	(* Falls nur Zentrierung aktiviert ist, dann zuerst den Schnellhub stoppen *)
	50:	IF NOT(xStFct_InitStep) THEN
			xStFct_InitStep:=TRUE;
			IF gxOnlyCentringActive OR (wStFct_Status = 99) OR (wStFct_Status = 1) OR (wStFct_Status = 98) THEN
				IF (T_Station_Parameter.T_StProcess.rCentringSpeedOAxis > 0.0) THEN
					QxFastStrokeOn_St1:=FALSE;
					QiAFastStroke:=0;
					TONWaitStopOAxis(IN:=FALSE,PT:=T#0.5s);
				ELSE
					TONWaitStopOAxis(IN:=FALSE,PT:=T#0.01s);
				END_IF;
			ELSE
				TONWaitStopOAxis(IN:=FALSE,PT:=T#0.01s);
			END_IF;
		END_IF;
		TONWaitStopOAxis(IN:=TRUE);
		IF TONWaitStopOAxis.Q THEN
			TONWaitStopOAxis(IN:=FALSE);
			xStFct_StartMainPrc:=FALSE;
			xStFct_InitStep:=FALSE;
			iStFct_StepPrc:=iStFct_StepPrc + 1;
		END_IF;
	(* Z1 Achse auf LadePosition zurückfahren ODER einen Offset zurückfahren *)
	51:	IF NOT(xStFct_InitStep) THEN
			xStFct_InitStep:=TRUE;
			IF gxOnlyCentringActive OR (wStFct_Status = 99) OR (wStFct_Status = 1) OR (wStFct_Status = 98) THEN
				ptrTAxisZ^.T_CtrleSingle.iFunction:=7;
				ptrTAxisZ^.T_CtrleSingle.lrPosition:=grZ_LoadPos;
				ptrTAxisZ^.T_CtrleSingle.lrVelocity:=T_Station_Parameter.T_StProcess.rOutfeedStrokeAxisSpeed;
				ptrTAxisZ^.T_CtrleSingle.xExecute:=TRUE;
				IF NOT(ptrTAxisBubbler^.T_CtrleDCAxis.xNotMoving) THEN
					(* Abstreifer ZU *)
					QxCylStripperClose_St1:=TRUE;
					QxCylStripperOpen_St1:=FALSE;
				END_IF
				IF (T_Station_Parameter.T_StProcess.rCentringSpeedOAxis > 0.0) THEN
					QxFastStrokeOn_St1:=FALSE;
					QiAFastStroke:=0;
				END_IF;
			ELSE
				lrZCheckPosition:=ptrTAxisZ^.T_LiveValue.lrActualPosition + T_Station_Parameter.T_StProcess.rCentringOffsetBackward;
				IF (lrZCheckPosition <= grZ_WorkStartPos) THEN
					ptrTAxisZ^.T_CtrleSingle.iFunction:=7;	(* Absolute Bewegung *)
					ptrTAxisZ^.T_CtrleSingle.lrPosition:=grZ_WorkStartPos;
				ELSE
					ptrTAxisZ^.T_CtrleSingle.iFunction:=8;	(* Relative Bewegung *)
					ptrTAxisZ^.T_CtrleSingle.lrDistance:=T_Station_Parameter.T_StProcess.rCentringOffsetBackward;
				END_IF;
				ptrTAxisZ^.T_CtrleSingle.lrVelocity:=T_Station_Parameter.T_StProcess.rCentringBackStrokeSpeed;
				ptrTAxisZ^.T_CtrleSingle.xExecute:=TRUE;
			END_IF;
		END_IF;
		IF (gxOnlyCentringActive OR (wStFct_Status = 99) OR (wStFct_Status = 1) OR (wStFct_Status = 98)) AND (ptrTAxisZ^.T_LiveValue.lrActualPosition <= (garCentringEndProcCalc[1] + T_Station_Parameter.T_StProcess.rCentringOffsetBackward)) THEN
			QxCylWPUnfix_St1:=FALSE;
		END_IF
		IF NOT(ptrTAxisZ^.T_CtrleSingle.xExecute) AND ptrTAxisZ^.T_CtrleSingle.xDone THEN
			xStFct_StartMainPrc:=FALSE;
			xStFct_InitStep:=FALSE;
			iStFct_StepPrc:=iStFct_StepPrc + 1;
			QxCylWPUnfix_St1:=FALSE;
		END_IF;
	(* S Achse stoppen *)
	(* O Achse stoppen *)
	(* ZylWPUnfix zurücksetzen *)
	52:	IF NOT(xStFct_InitStep) THEN
			xStFct_InitStep:=TRUE;
			IF gxOnlyCentringActive OR (wStFct_Status = 99) OR (wStFct_Status = 1) OR (wStFct_Status = 98) THEN
				IF (NOT(ptrTAxisS^.T_CtrleSingle.xNotMoving) OR NOT(ptrTAxisS^.T_CtrleSingle.xDone))
				AND NOT((ptrTAxisS^.T_CtrleSingle.iFunction = 5) AND NOT(ptrTAxisS^.T_CtrleSingle.xDone)) AND NOT(ptrTAxisS^.T_CtrleSingle.xErr) THEN
					ptrTAxisS^.T_CtrleSingle.iFunction:=5;
					ptrTAxisS^.T_CtrleSingle.xExecute:=TRUE;
				END_IF;
				IF (T_Station_Parameter.T_StProcess.rCentringSpeedOAxis > 0.0) THEN
					QxFastStrokeOn_St1:=FALSE;
					QiAFastStroke:=0;
				END_IF;
				QxCylWPUnfix_St1:=FALSE;
			END_IF
			IF xProcessDone THEN
				IF (NOT(ptrTAxisS^.T_CtrleSingle.xNotMoving) OR NOT(ptrTAxisS^.T_CtrleSingle.xDone))
				AND NOT((ptrTAxisS^.T_CtrleSingle.iFunction = 5) AND NOT(ptrTAxisS^.T_CtrleSingle.xDone)) AND NOT(ptrTAxisS^.T_CtrleSingle.xErr) THEN
					ptrTAxisS^.T_CtrleSingle.iFunction:=5;
					ptrTAxisS^.T_CtrleSingle.xExecute:=TRUE;
				END_IF;
				QxFastStrokeOn_St1:=FALSE;
				QiAFastStroke:=0;
			END_IF
			(* Abstreifer AUF *)
			QxCylStripperClose_St1:=FALSE;
			QxCylStripperOpen_St1:=TRUE;
		END_IF;
		IF NOT(ptrTAxisS^.T_CtrleSingle.xExecute) AND ptrTAxisS^.T_CtrleSingle.xDone THEN
			xStFct_StartMainPrc:=FALSE;
			xStFct_InitStep:=FALSE;
			IF (wStFct_Status <> 1) THEN
				iStFct_StepPrc:=90;
			ELSIF (wStFct_Status = 1) THEN
				xStFct_HardwareError:=TRUE;
				diStFct_TmpErrorNr:=41;		(* Zentrierproz. HC1 eingetroffen *)
				RETURN;
			ELSE
				xStFct_HardwareError:=TRUE;
				diStFct_TmpErrorNr:=42;		(* Zentrierproz. StartPos erreicht und HC2 immer noch ON *)
			END_IF;
		END_IF;

	90:	IF gxHardwareOFF OR gxAxisOFF THEN
		(* Gilt nur falls HW ausgeschaltet ist *)
			IF NOT(xStFct_InitStep) THEN
				xStFct_InitStep:=TRUE;
				TONWorkTime(IN:=FALSE);
			END_IF;
			TONWorkTime(IN:=TRUE,PT:=T#5s);
			T_Station_Work.THWWorkStation.TCtrlWork.iOverLimitCounterCentering:=5;
			IF TONWorkTime.Q THEN
				TONWorkTime(IN:=FALSE);
				xStFct_StartMainPrc:=FALSE;
				xStFct_InitStep:=FALSE;
				iStFct_StepPrc:=0;
				xStFct_SetEnd:=TRUE;
				wStFct_Status:=0;
				IF T_Station_Parameter.T_StProcess.xCentringEndProcIncOnOff THEN
					garCentringEndProcCalc[1]:=garCentringEndProcCalc[1] + T_Station_Parameter.T_StProcess.rCentringEndProInc;	(* Zentrier EndPos Inkrementieren *)
				END_IF;
			END_IF;
		ELSE
			xStFct_StartMainPrc:=FALSE;
			xStFct_InitStep:=FALSE;
			iStFct_StepPrc:=0;
			xStFct_SetEnd:=TRUE;
		END_IF;
	END_CASE;
END_IF;
(******************************************************************************************************************************************)
(****************************			             Stationsfunktion Parallelablauf                                       *****************************)
(******************************************************************************************************************************************)
IF xStFct_StartPrc_Parallel AND NOT(xStFct_SetEnd) AND NOT(xStFct_HardwareError) THEN
	CASE iStFct_StepPrc_Parallel OF
	1:	iStFct_StepPrc_Parallel:=1;
		xStFct_InitStep_Parallel:=FALSE;
		xStFct_StartPrc_Parallel:=FALSE;
	END_CASE;
END_IF;
(******************************************************************************************************************************************)
(****************************				     Stationsfunktion Endprozedur                                    *****************************)
(******************************************************************************************************************************************)
StationFunction_Ctrl_End;
END_ACTION

(* POU GENERAL/FB_CalcCuttingSpeed, ST *)
FUNCTION_BLOCK FB_CalcCuttingSpeed
VAR_INPUT
	rActualPosition : REAL;
	iCountStep : INT;	(* Durchschnitt von diesem Counter wird berechnet *)
END_VAR
VAR_IN_OUT
	xCapturePosition : BOOL;
	xReset : BOOL;
END_VAR
VAR_OUTPUT
	rCuttingSpeed : REAL;
END_VAR
VAR
	arCuttingSpeed: ARRAY [1..2,1..200] OF REAL;
	arDeleteData: ARRAY [1..2,1..200] OF REAL;
	iStepCounter: INT;
	rSumDeltaPos : REAL;
	rSumDeltaTime : REAL;
	ii: INT;
	iStepPos: INT;
	xFirstCycle: BOOL;
	rTmpSavePosition: REAL;
	TONCycleTime: TON;
	xStartTimer: BOOL;
	rTmpSaveTime: REAL;
	iTmpStepCount: INT;
END_VAR
(* Berechnung der Schnittgeschwindigkeit *)
IF xReset THEN
	xReset:=FALSE;
	xFirstCycle:=TRUE;
	xStartTimer:=FALSE;
	rCuttingSpeed:=0.0;
	arCuttingSpeed:=arDeleteData;
END_IF;
TONCycleTime(IN:=xStartTimer,PT:=T#999999s);
IF xCapturePosition THEN
	xCapturePosition:=xStartTimer:=FALSE;
	IF xFirstCycle THEN
		iTmpStepCount:=iCountStep;
		IF (iTmpStepCount <= 0) THEN
			iTmpStepCount:=1;
		ELSIF (iTmpStepCount > 200) THEN
			iTmpStepCount:=200;
		END_IF;
		xFirstCycle:=FALSE;
		iStepCounter:=iStepPos:=1;
		rCuttingSpeed:=0.0;
		rTmpSavePosition:=rActualPosition;
		xStartTimer:=TRUE;
		RETURN;
	END_IF;
	rTmpSavePosition:=rActualPosition - rTmpSavePosition;			(* Delta Position *)
	rTmpSaveTime:=TIME_TO_REAL(TONCycleTime.ET)/1000.0;		(* Delta Time *)
	arCuttingSpeed[1,iStepCounter]:=rTmpSavePosition;
	arCuttingSpeed[2,iStepCounter]:=rTmpSaveTime;
	rTmpSavePosition:=rActualPosition;
	rSumDeltaPos:=rSumDeltaTime:=0.0;
	FOR ii:=1 TO iStepPos DO
		rSumDeltaPos:=rSumDeltaPos + arCuttingSpeed[1,ii];
		rSumDeltaTime:=rSumDeltaTime + arCuttingSpeed[2,ii];
	END_FOR;
	rCuttingSpeed:=(rSumDeltaPos/INT_TO_REAL(iStepPos))/(rSumDeltaTime/INT_TO_REAL(iStepPos));
	iStepCounter:=iStepCounter + 1;
	IF (iStepCounter > iTmpStepCount) THEN
		iStepCounter:=1;
	END_IF;
	IF (iStepPos < iTmpStepCount) THEN
		iStepPos:=iStepPos + 1;
	END_IF;
ELSE
	IF NOT(xFirstCycle) THEN
		xStartTimer:=TRUE;
	END_IF;
END_IF;
END_FUNCTION_BLOCK

(* POU GENERAL/FB_SparkOutProcess, ST *)
FUNCTION_BLOCK FB_SparkOutProcess
VAR_INPUT
	lrHubLength: LREAL;
	iCountHub: INT;
	T_Station_Parameter: ST_RETAIN_DATA_STATIONWORK;
	xToolDeflection : BOOL;
	xToolTorqueHC : BOOL;
	xToolTorqueSparkOut : BOOL;
END_VAR
VAR_IN_OUT
	xStart: BOOL;
	xReset: BOOL;
	TCylToolDeflection : ST_CYLINDER;
	TAxisZ : ST_AXIS;
END_VAR
VAR_OUTPUT
	xEnd: BOOL;
	xBlockProcess: BOOL;
	xRepeatProcess: BOOL;
	wStatus: WORD;
	rLastOverLimitPosition: REAL;
	xBlockOutput:BOOL;
	xBlockDeflectionOutput:BOOL;
END_VAR
VAR
	xTmpStart: BOOL;
	xInit: BOOL;
	iStepCounter: INT;
	xInitStep: BOOL;
	lrSaveSlidePosition: LREAL;
	iTmpCountHub: INT;
	xSetForceDeflection: BOOL;
	xInitSetForceDeflection: BOOL;
	xActiveChgForceDeflection: BOOL;
	xBlockCounter: BOOL;
END_VAR
IF xReset THEN
	xReset:=FALSE;
	xEnd:=TRUE;
	xStart:=FALSE;
	xTmpStart:=FALSE;
	xInit:=FALSE;
	xBlockProcess:=FALSE;
	xRepeatProcess:=FALSE;
	xInitStep:=FALSE;
	iTmpCountHub:=0;
	xBlockOutput:=FALSE;
	RETURN;
END_IF;
IF xStart OR xTmpStart THEN
	IF NOT(xInit) THEN
		iStepCounter:=1;
		iTmpCountHub:=0;
		xInit:=TRUE;
		xStart:=FALSE;
		xTmpStart:=TRUE;
		lrSaveSlidePosition:=TAxisZ.T_LiveValue.lrActualPosition;
		xBlockProcess:=xRepeatProcess:=FALSE;
	END_IF;
	CASE iStepCounter OF
		1:	IF NOT(xInitStep) THEN
				xInitStep:=TRUE;
				xBlockProcess:=TRUE;
				xBlockCounter:=FALSE;
				IF (iCountHub > 0) AND (lrHubLength <> 0) THEN
					IF (T_Station_Parameter.T_StProcess.rSparkOutForceDeflection <> 0.0) THEN xActiveChgForceDeflection:=TRUE; ELSE xActiveChgForceDeflection:=FALSE; END_IF;
					IF NOT(xActiveChgForceDeflection) THEN
						xInitStep:=FALSE;
						iStepCounter:=iStepCounter + 1;
						RETURN;
					END_IF;
					IF xActiveChgForceDeflection THEN
						xBlockDeflectionOutput:=TRUE;
						xSetForceDeflection:=TRUE;
						TCylToolDeflection.T_CtrleCyl.T_Analog.rForceIn:=(T_Station_Parameter.T_OnlineChange.rForceDeflection/100.0) * T_Station_Parameter.T_StProcess.rSparkOutForceDeflection;
					ELSE
						xSetForceDeflection:=FALSE;
					END_IF;
				ELSE
					xEnd:=TRUE;
					xInit:=FALSE;
					xInitStep:=FALSE;
					xTmpStart:=FALSE;
					xBlockProcess:=xRepeatProcess:=xBlockOutput:=xBlockDeflectionOutput:=FALSE;
					RETURN;
				END_IF;
			END_IF;
			IF NOT(xSetForceDeflection) THEN
				xInitStep:=FALSE;
				iStepCounter:=iStepCounter + 1;
			END_IF;
		2:	IF NOT(xInitStep) THEN
				xInitStep:=TRUE;
				(* Move Absolut backward or forward *)
				TAxisZ.T_CtrleSingle.iFunction:=7;
				TAxisZ.T_CtrleSingle.lrPosition:=TAxisZ.T_LiveValue.lrActualPosition + lrHubLength;
				TAxisZ.T_CtrleSingle.lrAcceleration:=TAxisZ.T_Config_ObjFileValue.lrAcceleration;
				TAxisZ.T_CtrleSingle.lrDecceleration:=TAxisZ.T_Config_ObjFileValue.lrDecceleration;
				TAxisZ.T_CtrleSingle.lrJerk:=TAxisZ.T_Config_ObjFileValue.lrJerk;
				TAxisZ.T_CtrleSingle.lrVelocity:=T_Station_Parameter.T_StProcess.rSparkOutStrokeSpeed;
				TAxisZ.T_CtrleSingle.xExecute:=TRUE;
			END_IF;
			IF TAxisZ.T_CtrleSingle.xMovingForward THEN
				IF xToolDeflection THEN
					wStatus:=1;	(* 1 = < Wz Auslenk. Sensor > *)
					xInitStep:=FALSE;
					iStepCounter:=iStepCounter + 2;
					RETURN;
				END_IF;
				IF xToolTorqueHC THEN
					wStatus:=2;	(* 2 = < Wz Drehmom. HC> *)
					xInitStep:=FALSE;
					iStepCounter:=iStepCounter + 2;
					RETURN;
				END_IF
				IF xToolDeflection AND xToolTorqueHC THEN
					wStatus:=3;	(* 3 = < Wz Auslenk.+Wz Drehm.HC > *)
					xInitStep:=FALSE;
					iStepCounter:=iStepCounter + 2;
					RETURN;
				END_IF;
				IF xToolTorqueSparkOut THEN
					xBlockCounter:=TRUE;
				END_IF;
			END_IF;
			IF NOT(TAxisZ.T_CtrleSingle.xExecute) AND TAxisZ.T_CtrleSingle.xDone THEN
				xInitStep:=FALSE;
				iStepCounter:=iStepCounter + 1;
			END_IF;
		3:	IF NOT(xInitStep) THEN
				xInitStep:=TRUE;
				(* Move Absolut forward or backward *)
				TAxisZ.T_CtrleSingle.iFunction:=7;
				TAxisZ.T_CtrleSingle.lrPosition:=lrSaveSlidePosition;
				TAxisZ.T_CtrleSingle.lrAcceleration:=TAxisZ.T_Config_ObjFileValue.lrAcceleration;
				TAxisZ.T_CtrleSingle.lrDecceleration:=TAxisZ.T_Config_ObjFileValue.lrDecceleration;
				TAxisZ.T_CtrleSingle.lrJerk:=TAxisZ.T_Config_ObjFileValue.lrJerk;
				TAxisZ.T_CtrleSingle.lrVelocity:=T_Station_Parameter.T_StProcess.rSparkOutStrokeSpeed;
				TAxisZ.T_CtrleSingle.xExecute:=TRUE;
			END_IF;
			IF TAxisZ.T_CtrleSingle.xMovingForward THEN
				IF xToolDeflection THEN
					wStatus:=1;	(* 1 = < Wz Auslenk. Sensor > *)
					xInitStep:=FALSE;
					iStepCounter:=iStepCounter + 1;
					RETURN;
				END_IF;
				IF xToolTorqueHC THEN
					wStatus:=2;	(* 2 = < Wz Drehmom. HC> *)
					xInitStep:=FALSE;
					iStepCounter:=iStepCounter + 1;
					RETURN;
				END_IF
				IF xToolDeflection AND xToolTorqueHC THEN
					wStatus:=3;	(* 3 = < Wz Auslenk.+Wz Drehm.HC > *)
					xInitStep:=FALSE;
					iStepCounter:=iStepCounter + 1;
					RETURN;
				END_IF;
				IF xToolTorqueSparkOut THEN
					xBlockCounter:=TRUE;
				END_IF;
			END_IF;
			IF NOT(TAxisZ.T_CtrleSingle.xExecute) AND TAxisZ.T_CtrleSingle.xDone THEN
				IF NOT(xBlockCounter) THEN
					iTmpCountHub:=iTmpCountHub + 1;
				END_IF;
				xBlockCounter:=FALSE;
				IF (iTmpCountHub >= iCountHub) THEN
					IF NOT(xActiveChgForceDeflection) THEN
						xEnd:=TRUE;
						xInit:=FALSE;
						xInitStep:=FALSE;
						xTmpStart:=FALSE;
						xBlockProcess:=xRepeatProcess:=xBlockOutput:=xBlockDeflectionOutput:=FALSE;
					ELSE
						xInitStep:=FALSE;
						iStepCounter:=5;
					END_IF;
				ELSE
					xInitStep:=FALSE;
					iStepCounter:=2;
				END_IF;
			END_IF;
		4:	IF NOT(xInitStep) THEN
				xInitStep:=TRUE;
				IF NOT(TAxisZ.T_CtrleSingle.xNotMoving) THEN
					rLastOverLimitPosition:=TAxisZ.T_LiveValue.lrActualPosition;
					TAxisZ.T_CtrleSingle.iFunction:=5;
					TAxisZ.T_CtrleSingle.xExecute:=TRUE;
					RETURN;
				END_IF
				IF NOT(TAxisZ.T_CtrleSingle.xDone) THEN
					xInitStep:=FALSE;
					RETURN;
				END_IF;
			END_IF;
			IF NOT(TAxisZ.T_CtrleSingle.xExecute) AND TAxisZ.T_CtrleSingle.xDone THEN
				IF NOT(xActiveChgForceDeflection) THEN
					xRepeatProcess:=TRUE;
					xEnd:=TRUE;
					xInit:=FALSE;
					xInitStep:=FALSE;
					xTmpStart:=FALSE;
					xBlockProcess:=FALSE;
					xBlockOutput:=FALSE;
					xBlockDeflectionOutput:=FALSE;
				ELSE
					xInitStep:=FALSE;
					iStepCounter:=6;
				END_IF;
			END_IF;
		5:	IF NOT(xInitStep) THEN
				xInitStep:=TRUE;
				IF xActiveChgForceDeflection THEN
					xSetForceDeflection:=TRUE;
					xBlockDeflectionOutput:=TRUE;
					TCylToolDeflection.T_CtrleCyl.T_Analog.rForceIn:=T_Station_Parameter.T_OnlineChange.rForceDeflection;
				ELSE
					xSetForceDeflection:=FALSE;
				END_IF;
			END_IF;
			IF NOT(xSetForceDeflection) THEN
				xBlockOutput:=FALSE;
				xBlockDeflectionOutput:=FALSE;
				xEnd:=TRUE;
				xInit:=FALSE;
				xInitStep:=FALSE;
				xTmpStart:=FALSE;
				xBlockProcess:=xRepeatProcess:=FALSE;
			END_IF;
		6:	IF NOT(xInitStep) THEN
				xInitStep:=TRUE;
				IF xActiveChgForceDeflection THEN
					xSetForceDeflection:=TRUE;
					xBlockDeflectionOutput:=TRUE;
					TCylToolDeflection.T_CtrleCyl.T_Analog.rForceIn:=T_Station_Parameter.T_OnlineChange.rForceDeflection;
				ELSE
					xSetForceDeflection:=FALSE;
				END_IF;
			END_IF;
			IF NOT(xSetForceDeflection) THEN
				xBlockOutput:=FALSE;
				xBlockDeflectionOutput:=FALSE;
				xRepeatProcess:=TRUE;
				xEnd:=TRUE;
				xInit:=FALSE;
				xInitStep:=FALSE;
				xTmpStart:=FALSE;
				xBlockProcess:=FALSE;
			END_IF;
	END_CASE;

	IF xSetForceDeflection THEN
		IF NOT(xInitSetForceDeflection) THEN
			IF NOT(TCylToolDeflection.T_CtrleCyl.xExecute) AND TCylToolDeflection.T_CtrleCyl.xDone THEN
				xInitSetForceDeflection:=TRUE;
				TCylToolDeflection.T_CtrleCyl.iFunction:=4;
				TCylToolDeflection.T_CtrleCyl.xExecute:=TRUE;
			END_IF;
		END_IF;
		IF NOT(TCylToolDeflection.T_CtrleCyl.xExecute) AND TCylToolDeflection.T_CtrleCyl.xDone AND xInitSetForceDeflection THEN
			xInitSetForceDeflection:=FALSE;
			xSetForceDeflection:=FALSE;
		END_IF;
	END_IF;
ELSE
	xBlockOutput:=FALSE;
	xBlockDeflectionOutput:=FALSE;
END_IF;
END_FUNCTION_BLOCK

(* POU GENERAL/FB_PID_CONTROL, ST *)
FUNCTION_BLOCK FB_PID_CONTROL
VAR_INPUT
	rSetpointValue    : REAL;
    rActualValue      : REAL;
END_VAR
VAR_IN_OUT
	T_CtrlPara:ST_CTRL_PID_PARAM;
END_VAR
VAR_OUTPUT
	rOut:REAL;
	xMaxOutputReach:BOOL;
	xMinOutputReach:BOOL;
END_VAR
VAR
	r_E_Fehler:REAL;
	r_E_Fehler_Sum:REAL;
	r_E_Fehler_Alt:REAL;
	r_Zykluszeit:REAL;
	r_P_Anteil:REAL;
	r_I_Anteil:REAL;
	r_D_Anteil:REAL;
	TONWaitMinTime: TON;
END_VAR
r_E_Fehler:=rSetpointValue - rActualValue;	(* Regelabweichung *)
IF NOT(xMaxOutputReach) AND NOT(xMinOutputReach) THEN
	r_E_Fehler_Sum:=r_E_Fehler_Sum + r_E_Fehler;
END_IF
r_Zykluszeit:=T_CtrlPara.rCtrlCycleTime;
IF (r_Zykluszeit = 0.0) THEN
	r_Zykluszeit:=0.001;
END_IF
r_P_Anteil:=T_CtrlPara.rKp * r_E_Fehler;
r_I_Anteil:=T_CtrlPara.rKi * r_Zykluszeit * r_E_Fehler_Sum;
r_D_Anteil:=(T_CtrlPara.rKd/r_Zykluszeit) * (r_E_Fehler - r_E_Fehler_Alt);
rOut:=r_P_Anteil + r_I_Anteil + r_D_Anteil;
r_E_Fehler_Alt:=r_E_Fehler;
IF (rOut >= T_CtrlPara.rOutMaxLimit) THEN
	rOut:=T_CtrlPara.rOutMaxLimit;
	xMaxOutputReach:=TRUE;
ELSE
	xMaxOutputReach:=FALSE;
END_IF
IF (rOut <= T_CtrlPara.rOutMinLimit) THEN
	rOut:=T_CtrlPara.rOutMinLimit;
	TONWaitMinTime(IN:=TRUE,PT:=T#100MS);
	IF TONWaitMinTime.Q THEN
		xMinOutputReach:=TRUE;	(* Das Minimum muss mindestens 100ms anstehen, damit dieser Ausgang gesetzt wird. Dies veranlasst dann ein HC, da die minimale Geschwindigkeit erreicht ist *)
	END_IF;
ELSE
	TONWaitMinTime(IN:=FALSE);
	xMinOutputReach:=FALSE;
END_IF
IF T_CtrlPara.xReset_I_Anteil THEN
	T_CtrlPara.xReset_I_Anteil:=FALSE;
	r_E_Fehler_Sum:=0.0;
END_IF
END_FUNCTION_BLOCK

(* POU GENERAL/FB_D_CONTROL, ST *)
FUNCTION_BLOCK FB_D_CONTROL
VAR_INPUT
    rActualValue      : REAL;
END_VAR
VAR_IN_OUT
	T_CtrlPara:ST_CTRL_PID_PARAM;
END_VAR
VAR_OUTPUT
	rOut:REAL;
	xMaxOutputReach:BOOL;
	xMinOutputReach:BOOL;
END_VAR
VAR
	r_E_Fehler:REAL;
	r_E_Fehler_Alt:REAL;
	r_Zykluszeit:REAL;
	r_D_Anteil:REAL;
END_VAR
(* Es wird nur eine Ausgabe bei Abweichung zwischen vorgehendem und aktuellen Wert berechnet *)
r_E_Fehler:= rActualValue;
r_Zykluszeit:=T_CtrlPara.rCtrlCycleTime;
IF (r_Zykluszeit = 0.0) THEN
	r_Zykluszeit:=0.001;
END_IF
r_D_Anteil:=(T_CtrlPara.rKd/r_Zykluszeit) * (r_E_Fehler - r_E_Fehler_Alt);
rOut:=r_D_Anteil;
r_E_Fehler_Alt:=r_E_Fehler;
IF (rOut >= T_CtrlPara.rOutMaxLimit) THEN
	rOut:=T_CtrlPara.rOutMaxLimit;
	xMaxOutputReach:=TRUE;
ELSE
	xMaxOutputReach:=FALSE;
END_IF
IF (rOut <= T_CtrlPara.rOutMinLimit) THEN
	rOut:=T_CtrlPara.rOutMinLimit;
	xMinOutputReach:=TRUE;
ELSE
	xMinOutputReach:=FALSE;
END_IF
END_FUNCTION_BLOCK

(* POU PRG_COLLISION_DETECTION, ST *)
PROGRAM PRG_COLLISION_DETECTION
VAR
	ptrTCommonStation:POINTER TO ST_STATION;
	ptrTCommonStation0:POINTER TO ST_STATION;
	ptrTCommonAxis : POINTER TO ST_AXIS;
	ptrTCommonAxis0 : POINTER TO ST_AXIS;
	xTmp: BOOL;
	xTmp0: BOOL;
	xActiveMessageWork: BOOL;
	xActiveMessageWork1: BOOL;
	xCheckHCSensor: BOOL;
	xCheckZAxisVelModePosDirection: BOOL;
	xCheckMovement: BOOL;
	xCheckZAxisRelPosDirection: BOOL;
	xCheckZAxisAbsPosDirection: BOOL;
	iSaveAxisNr:INT;
	diSaveAxisZErrNr: DINT;
	diSaveAxisZErr1Nr: DINT;
	ii: INT;
	xZAxisBrakeReleased: BOOL;
	xCheckHCOverloadSensor: BOOL;
	jj: INT;
	iSaveStateMessage: INT;
	TONCheckRelease: TON;
END_VAR
(* Kollisionsüberprüfung für den HandBetrieb und Prozess *)
	Check_Station_Working_AxisBrake;
	Check_Station_Working;
END_PROGRAM
ACTION Check_Station_Working:
IF NOT(T_StartUp.T_State.xCompleted) OR gxHardwareOFF OR gxAxisOFF THEN
	RETURN;
END_IF;
(* Überprüfe den Zustand der Zylinder *)
(* Überwachung im AutoBetrieb und HandBetrieb *)
IF NOT(TProcess.T_Ctrle.xExecute) AND TProcess.T_Ctrle.xDone AND NOT(TProcess.T_Ctrle.xError) OR TRUE THEN
(* Zylinder Überwachung der Bearbeitungsstation MicroHead und Entgrat *)
(* Achsen Überwachung der Bearbeitungsstation MicroHead und Entgrat *)
	FOR ii:=1 TO 1 DO
		IF (ii = 1) THEN ptrTCommonStation:=ADR(TStation_Work_St1); jj:=1; END_IF;
		ptrTCommonAxis:=ADR(ptrTCommonStation^.THWWorkStation.TAxisZ);
		xCheckHCSensor:=			ptrTCommonStation^.THWWorkStation.TCylToolDeflection.T_CtrleCyl.xStatePosOn AND NOT(ptrTCommonStation^.TControl.xExecute) AND ptrTCommonStation^.TControl.xDone AND
									NOT(ptrTCommonStation^.TControl.xError) AND ptrTCommonStation^.TControl.xRdy;
		xCheckHCOverloadSensor:=	FALSE;
		(* Für Z Achse muss die Positive Richtung für HC überprüft werden *)
		xCheckZAxisVelModePosDirection:=(ptrTCommonAxis^.T_CtrleSingle.iFunction = 6) AND (ptrTCommonAxis^.T_CtrleSingle.lrVelocity >= 0);
		xCheckZAxisRelPosDirection:=(ptrTCommonAxis^.T_CtrleSingle.iFunction = 8) AND (ptrTCommonAxis^.T_CtrleSingle.lrDistance >= 0);
		xCheckZAxisAbsPosDirection:=(ptrTCommonAxis^.T_CtrleSingle.iFunction = 7) AND (ptrTCommonAxis^.T_CtrleSingle.lrPosition > ptrTCommonAxis^.T_LiveValue.lrActualPosition);
		xCheckMovement:=	(xCheckHCSensor OR xCheckHCOverloadSensor) AND
							(xCheckZAxisVelModePosDirection OR xCheckZAxisRelPosDirection OR xCheckZAxisAbsPosDirection);
		IF ptrTCommonAxis^.T_CtrleSingle.xExecute AND ptrTCommonAxis^.T_CtrleSingle.xDone THEN
			(* Überprüfung für Achse wenn Start Befehl erfolgt *)
			xTmp:=	xCheckMovement;
			IF xTmp THEN
				(* Überprüfe nun ob die Achse sich bewegen darf *)
				IF (ptrTCommonAxis^.T_CtrleSingle.iFunction <> 1) AND (ptrTCommonAxis^.T_CtrleSingle.iFunction <> 3) AND (ptrTCommonAxis^.T_CtrleSingle.iFunction <> 4) THEN
					ptrTCommonAxis^.T_CtrleSingle.xExecute:=FALSE;		(* Aufruf des Aktuators wird zurückgesetzt *)
					T_VisuQVis.T_CtrleAction.xDeleteVisuFunction:=TRUE;
					T_VisuQVis.T_CtrleAction.xFunctionActive:=FALSE;
					xActiveMessageWork1:=TRUE;
					IF xCheckHCSensor THEN
						iSaveStateMessage:=241;		(* Warnung: Kollisionsgefahr: WzAuslenkung Sensor ST1 Aktiv ! *)
					ELSIF xCheckHCOverloadSensor THEN
						iSaveStateMessage:=245;		(* Warnung: Kollisionsgefahr: WzDrehmoment Überlast Sensor ST1 Aktiv ! *)
					END_IF;
				END_IF;
			END_IF;
		END_IF;
		IF NOT(ptrTCommonAxis^.T_CtrleSingle.xNotMoving) AND NOT(ptrTCommonAxis^.T_CtrleSingle.xExecute) AND (ptrTCommonAxis^.T_CtrleSingle.iFunction <> 5) THEN
			(* Überprüfung für Achse wenn sich in Positiver Richtung bewegt *)
			IF ptrTCommonAxis^.T_CtrleSingle.xMovingForward THEN
				(* Überprüfe nun ob die Achse gestoppt werden muss *)
				IF xCheckMovement THEN
					(* Teller liegt nicht im Raster, daher muss die Achse gestoppt werden *)
					ptrTCommonAxis^.T_CtrleSingle.iFunction:=5;
					ptrTCommonAxis^.T_CtrleSingle.xExecute:=TRUE;
					T_VisuQVis.T_CtrleAction.xDeleteVisuFunction:=TRUE;
					T_VisuQVis.T_CtrleAction.xFunctionActive:=FALSE;
					xActiveMessageWork1:=TRUE;
					IF xCheckHCSensor THEN
						iSaveStateMessage:=241;		(* Warnung: Kollisionsgefahr: WzAuslenkung Sensor ST1 Aktiv ! *)
					ELSIF xCheckHCOverloadSensor THEN
						iSaveStateMessage:=245;		(* Warnung: Kollisionsgefahr: WzDrehmoment Überlast Sensor ST1 Aktiv ! *)
					END_IF;
				END_IF;
			END_IF;
		END_IF;
	END_FOR;

	IF xActiveMessageWork1 THEN
		xActiveMessageWork1:=FALSE;
		T_ExchgParam.T_Visu.T_Message.iState:=iSaveStateMessage;
	ELSE
		diSaveAxisZErr1Nr:=0;
	END_IF;
END_IF;
END_ACTION
ACTION Check_Station_Working_AxisBrake:
IF NOT(T_StartUp.T_State.xCompleted) OR gxHardwareOFF THEN
	RETURN;
END_IF;
(* Überprüfe den Zustand der Zylinder *)
TONCheckRelease(IN:=NOT(TStation_Work_St1.THWWorkStation.TCylBrakeReleaseZAxis.T_CtrleCyl.xStatePosOn), PT:=T#1S);
IF TStation_Work_St1.THWWorkStation.TCylBrakeReleaseZAxis.T_CtrleCyl.xStatePosOn THEN
	TCollisionDetection.xZAxisBrakeReleased:=TRUE;	(* Bremse gelöst *)
END_IF;
IF TONCheckRelease.Q THEN
	TCollisionDetection.xZAxisBrakeReleased:=FALSE;	(* Bremse nicht gelöst *)
END_IF;

(* Überwachung im AutoBetrieb und HandBetrieb *)
IF NOT(TProcess.T_Ctrle.xExecute) AND TProcess.T_Ctrle.xDone AND NOT(TProcess.T_Ctrle.xError) OR TRUE THEN
(* Achsen Überwachung der Bearbeitungsstation MicroHead *)
	FOR ii:=1 TO 1 DO
		IF (ii = 1) THEN ptrTCommonStation0:=ADR(TStation_Work_St1); xZAxisBrakeReleased:=TCollisionDetection.xZAxisBrakeReleased;END_IF;
		ptrTCommonAxis0:=ADR(ptrTCommonStation0^.THWWorkStation.TAxisZ);
		IF ptrTCommonAxis0^.T_CtrleSingle.xExecute AND ptrTCommonAxis0^.T_CtrleSingle.xDone THEN
			(* Überprüfung für Achse wenn Start Befehl erfolgt *)
			xTmp0:=	(ptrTCommonAxis0^.T_CtrleSingle.iFunction = 6) OR (ptrTCommonAxis0^.T_CtrleSingle.iFunction = 7) OR (ptrTCommonAxis0^.T_CtrleSingle.iFunction = 8) OR (ptrTCommonAxis0^.T_CtrleSingle.iFunction = 9);
			IF xTmp0 THEN
				(* Überprüfe nun ob die Achse sich bewegen darf *)
				IF NOT(xZAxisBrakeReleased) AND NOT(ptrTCommonAxis0^.T_CtrleSingle.xStateHWLimitPos) AND NOT(ptrTCommonAxis0^.T_CtrleSingle.xStateHWLimitNeg) THEN
					(* Bremse ist Aktiv und deshalb darf die Achse nicht verfahren werden *)
					ptrTCommonAxis0^.T_CtrleSingle.xExecute:=FALSE;		(* Aufruf des Aktuators wird zurückgesetzt *)
					T_VisuQVis.T_CtrleAction.xDeleteVisuFunction:=TRUE;
					T_VisuQVis.T_CtrleAction.xFunctionActive:=FALSE;
					xActiveMessageWork:=TRUE;
					iSaveAxisNr:=ii;
				END_IF;
			END_IF;
		END_IF;
		IF NOT(ptrTCommonAxis0^.T_CtrleSingle.xNotMoving) AND NOT(ptrTCommonAxis0^.T_CtrleSingle.xExecute) AND (ptrTCommonAxis0^.T_CtrleSingle.iFunction <> 5) THEN
			(* Überprüfe nun ob die Achse gestoppt werden muss *)
			IF NOT(xZAxisBrakeReleased) AND NOT(ptrTCommonAxis0^.T_CtrleSingle.xStateHWLimitPos) AND NOT(ptrTCommonAxis0^.T_CtrleSingle.xStateHWLimitNeg) THEN
				(* Teller liegt nicht im Raster, daher muss die Achse gestoppt werden *)
				ptrTCommonAxis0^.T_CtrleSingle.iFunction:=5;
				ptrTCommonAxis0^.T_CtrleSingle.xExecute:=TRUE;
				T_VisuQVis.T_CtrleAction.xDeleteVisuFunction:=TRUE;
				T_VisuQVis.T_CtrleAction.xFunctionActive:=FALSE;
				xActiveMessageWork:=TRUE;
				iSaveAxisNr:=ii;
			END_IF;
		END_IF;
	END_FOR;
	IF xActiveMessageWork THEN
		xActiveMessageWork:=FALSE;
		IF (iSaveAxisNr = 1) THEN
			T_ExchgParam.T_Visu.T_Message.iState:=239;		(* Warnung: Kollisionsgefahr: Z Achse ST1 Bremse Aktiv ! *)
			ptrTCommonStation0:=ADR(TStation_Work_St1);
		END_IF;
		ptrTCommonAxis0:=ADR(ptrTCommonStation0^.THWWorkStation.TAxisZ);
		IF NOT(ptrTCommonStation0^.TControl.xExecute) AND NOT(ptrTCommonStation0^.TControl.xDone) AND NOT(ptrTCommonStation0^.TControl.xError) THEN
			IF (diSaveAxisZErrNr = 0) THEN
				IF (T_ExchgParam.T_Visu.T_Message.iState = 239) THEN
					diSaveAxisZErrNr:=16#F501;		(* Bremse Aktiv von ST1 *)
				ELSIF (T_ExchgParam.T_Visu.T_Message.iState = 240) THEN
					diSaveAxisZErrNr:=16#F502;		(* Bremse Aktiv von ST2 *)
				ELSIF (T_ExchgParam.T_Visu.T_Message.iState = 255) THEN
					diSaveAxisZErrNr:=16#F503;		(* Bremse Aktiv von ST3 *)
				ELSIF (T_ExchgParam.T_Visu.T_Message.iState = 256) THEN
					diSaveAxisZErrNr:=16#F504;		(* Bremse Aktiv von ST4 *)
				END_IF;
			END_IF;
			IF NOT(ptrTCommonAxis0^.T_CtrleSingle.xExecute) AND ptrTCommonAxis0^.T_CtrleSingle.xDone AND
			     NOT(ptrTCommonAxis0^.T_CtrleSingle.xErr) AND ptrTCommonAxis0^.T_CtrleSingle.xNotMoving THEN
				ptrTCommonAxis0^.T_CtrleSingle.xErr:=TRUE;
				ptrTCommonAxis0^.T_CtrleSingle.xDone:=FALSE;
				ptrTCommonAxis0^.T_CtrleSingle.udiErrorID:=diSaveAxisZErrNr;
			ELSE
				xActiveMessageWork:=TRUE;
			END_IF;
		END_IF;
	ELSE
		diSaveAxisZErrNr:=0;
	END_IF;
END_IF;
END_ACTION

(* POU PRG_VELOCITY_DETECTION, ST *)
PROGRAM PRG_VELOCITY_DETECTION
VAR
	ptrTCommonAxis : POINTER TO ST_AXIS;
	xTmp: BOOL;
	lrSaveZAxisVelocity: LREAL;
	lrMaxVelocity_Z_Axis: LREAL;
	xSLS_Z_Axis: BOOL;
	lrMaxVelocity_SetupA_Z_Axis:LREAL:=79.0;
	lrMaxVelocity_SetupB_Z_Axis:LREAL:=29.9;
END_VAR
Check_Station_Working;
gxSetSpeedInMovement:=FALSE;
END_PROGRAM
ACTION Check_Station_Working:
IF gT_SafetyStatus.xSetupOperateModeActive THEN
	ptrTCommonAxis:=ADR(TStation_Work_St1.THWWorkStation.TAxisZ);
	IF (gT_SafetyStatus.iSetupMode = 1) THEN
		lrMaxVelocity_Z_Axis:=lrMaxVelocity_SetupA_Z_Axis;
		xSLS_Z_Axis:=T_TwinSafe_Status_Z_Axis_St1.xSLS1;
	ELSIF (gT_SafetyStatus.iSetupMode = 2) THEN
		lrMaxVelocity_Z_Axis:=lrMaxVelocity_SetupB_Z_Axis;
		xSLS_Z_Axis:=T_TwinSafe_Status_Z_Axis_St1.xSLS2;
	ELSE
		lrMaxVelocity_Z_Axis:=lrMaxVelocity_SetupA_Z_Axis;
		xSLS_Z_Axis:=T_TwinSafe_Status_Z_Axis_St1.xSLS1;
	END_IF;
	IF gT_SafetyStatus.xSecurityDoorOpen THEN
		xTmp:=	ptrTCommonAxis^.T_CtrleSingle.xExecute AND ptrTCommonAxis^.T_CtrleSingle.xDone AND ptrTCommonAxis^.T_CtrleSingle.xNotMoving AND
				((ptrTCommonAxis^.T_CtrleSingle.iFunction = 6) OR (ptrTCommonAxis^.T_CtrleSingle.iFunction = 7) OR (ptrTCommonAxis^.T_CtrleSingle.iFunction = 8));
		IF xTmp THEN
			IF (ABS(ptrTCommonAxis^.T_CtrleSingle.lrVelocity) >= lrMaxVelocity_Z_Axis) THEN
				lrSaveZAxisVelocity:=ptrTCommonAxis^.T_CtrleSingle.lrVelocity;
				IF (lrSaveZAxisVelocity >= 0) THEN
					ptrTCommonAxis^.T_CtrleSingle.lrVelocity:=lrMaxVelocity_Z_Axis - 0.1;
				ELSE
					ptrTCommonAxis^.T_CtrleSingle.lrVelocity:=(lrMaxVelocity_Z_Axis - 0.1) * -1.0;
				END_IF;
			END_IF;
		END_IF;
		xTmp:=	NOT(ptrTCommonAxis^.T_CtrleSingle.xExecute) AND ptrTCommonAxis^.T_CtrleSingle.xDone AND NOT(ptrTCommonAxis^.T_CtrleSingle.xNotMoving) AND (ptrTCommonAxis^.T_CtrleSingle.iFunction = 6);
		xTmp:=	xTmp OR (NOT(ptrTCommonAxis^.T_CtrleSingle.xExecute) AND NOT(ptrTCommonAxis^.T_CtrleSingle.xDone) AND NOT(ptrTCommonAxis^.T_CtrleSingle.xNotMoving) AND
				((ptrTCommonAxis^.T_CtrleSingle.iFunction = 7) OR (ptrTCommonAxis^.T_CtrleSingle.iFunction = 8))) OR gxSetSpeedInMovement;
		IF xTmp THEN
			IF (ABS(ptrTCommonAxis^.T_CtrleSingle.lrVelocity) >= lrMaxVelocity_Z_Axis) THEN
				lrSaveZAxisVelocity:=ptrTCommonAxis^.T_CtrleSingle.lrVelocity;
				ptrTCommonAxis^.T_CtrleSingle.lrVelocity:=lrMaxVelocity_Z_Axis - 0.1;
				ptrTCommonAxis^.T_CtrleSingle.iFunction:=12;
				ptrTCommonAxis^.T_CtrleSingle.xExecute:=TRUE;
			END_IF;
		END_IF;
	ELSE
		xTmp:=	NOT(ptrTCommonAxis^.T_CtrleSingle.xExecute) AND ptrTCommonAxis^.T_CtrleSingle.xDone AND NOT(ptrTCommonAxis^.T_CtrleSingle.xNotMoving) AND (ptrTCommonAxis^.T_CtrleSingle.iFunction = 6);
		xTmp:=	xTmp OR (NOT(ptrTCommonAxis^.T_CtrleSingle.xExecute) AND NOT(ptrTCommonAxis^.T_CtrleSingle.xDone) AND NOT(ptrTCommonAxis^.T_CtrleSingle.xNotMoving) AND
				((ptrTCommonAxis^.T_CtrleSingle.iFunction = 7) OR (ptrTCommonAxis^.T_CtrleSingle.iFunction = 8)));
		IF xTmp THEN
			IF (ptrTCommonAxis^.T_CtrleSingle.lrVelocity <> lrSaveZAxisVelocity) AND (lrSaveZAxisVelocity <> 0) AND NOT(xSLS_Z_Axis) THEN
				ptrTCommonAxis^.T_CtrleSingle.lrVelocity:=lrSaveZAxisVelocity;
				ptrTCommonAxis^.T_CtrleSingle.iFunction:=12;
				ptrTCommonAxis^.T_CtrleSingle.xExecute:=TRUE;
			END_IF;
		END_IF;
	END_IF;
	IF (NOT(ptrTCommonAxis^.T_CtrleSingle.xExecute) AND ptrTCommonAxis^.T_CtrleSingle.xDone AND ptrTCommonAxis^.T_CtrleSingle.xNotMoving) OR ptrTCommonAxis^.T_CtrleSingle.xErr THEN
		lrSaveZAxisVelocity:=0.0;
	END_IF;
END_IF;
END_ACTION

(* POU PRG_LAYER2_HARDWARE/PRG_HW_WORK_ST1, FBD *)
PROGRAM PRG_HW_WORK_ST1
VAR
	FBHWStationWork_St1: FBHW_STATION_WORK;
(* Axis value *)
	IuiActualTorqueAxisZ_St1 AT %I*:UINT;
	IwInputState_Z_Axis_St1 AT %I*:WORD;
	IuiActualTorqueAxisS_St1 AT %I*:UINT;
	IwInputState_S1_Axis_St1 AT %I*:WORD;
	IwInputState_S2_Axis_St1 AT %I*:WORD;									(* IGS *)
	IwInputState_S3_Axis_St1 AT %I*:WORD;									(* IGS *)

(* Axis structure *)
	stZRefIn_St1 AT %I* :NCTOPLC_AXLESTRUCT;
	stZRefOut_St1 AT %Q* :PLCTONC_AXLESTRUCT;
	stZDriveState_St1 AT %I*:ST_AXIS_DRIVESTATE;
	stSRefIn_St1 AT %I* :NCTOPLC_AXLESTRUCT;
	stSRefOut_St1 AT %Q* :PLCTONC_AXLESTRUCT;
	stS2RefIn_St1 AT %I* :NCTOPLC_AXLESTRUCT;		(* Beckhoff Spindel L *)	(* IGS *)
	stS2RefOut_St1 AT %Q* :PLCTONC_AXLESTRUCT;	(* Beckhoff Spindel L *)	(* IGS *)
	stS3RefIn_St1 AT %I* :NCTOPLC_AXLESTRUCT;		(* Beckhoff Spindel M *)	(* IGS *)
	stS3RefOut_St1 AT %Q* :PLCTONC_AXLESTRUCT;	(* Beckhoff Spindel M *)	(* IGS *)

(* Axis DC structure *)
	stBubblerDataINSt1 AT %I*  : ST_COMM_IN_DCAXIS;			(* IGS3 *)
	stBubblerDataOUTSt1 AT %Q*  : ST_COMM_OUT_DCAXIS;		(* IGS3 *)
	stFeedpumpINDataSt1 AT %I*  : ST_COMM_IN_DCAXIS;		(* IGS3 *)
	stFeedpumpOUTDataSt1 AT %Q*  : ST_COMM_OUT_DCAXIS;	(* IGS3 *)

(* FB Output *)
	xActiveHWWork_St1 : BOOL;
	xActiveStationWork_St1 : BOOL;
	wState_Z_Axis_St1: WORD;

	xStationPowerON_St1:BOOL;

(* Drehmomentüberlast *)
	IudiTorqueOverloadCounterValue_St1			AT%I*:UDINT;	(* Clock-->Signal induktiver Sensor für Drehmomentüberlast *)		(* IGS *)
END_VAR
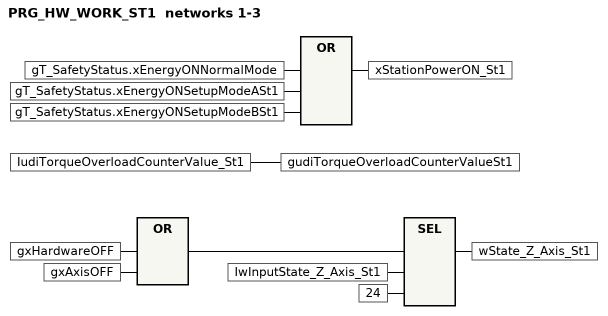
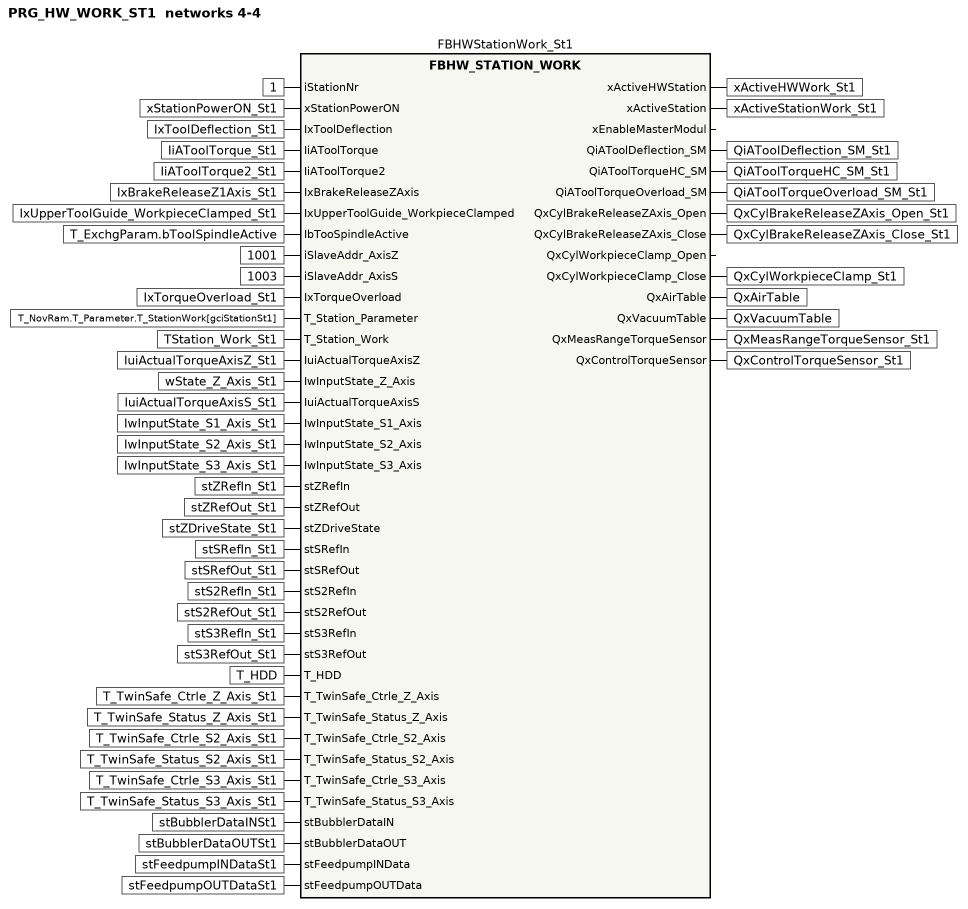
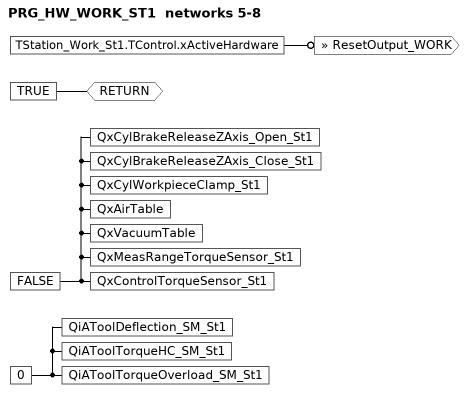
_FBD_ (* Function Block Diagram *)
NETWORK 1
	OR(gT_SafetyStatus.xEnergyONNormalMode, gT_SafetyStatus.xEnergyONSetupModeASt1, gT_SafetyStatus.xEnergyONSetupModeBSt1) => xStationPowerON_St1
NETWORK 2
	IudiTorqueOverloadCounterValue_St1 => gudiTorqueOverloadCounterValueSt1
NETWORK 3
	SEL(OR(gxHardwareOFF, gxAxisOFF), IwInputState_Z_Axis_St1, 24) => wState_Z_Axis_St1
NETWORK 4
	FBHWStationWork_St1:FBHW_STATION_WORK(iStationNr: 1, xStationPowerON: xStationPowerON_St1, IxToolDeflection: IxToolDeflection_St1, IiAToolTorque: IiAToolTorque_St1, IiAToolTorque2: IiAToolTorque2_St1, IxBrakeReleaseZAxis: IxBrakeReleaseZ1Axis_St1, IxUpperToolGuide_WorkpieceClamped: IxUpperToolGuide_WorkpieceClamped_St1, IbTooSpindleActive: T_ExchgParam.bToolSpindleActive, iSlaveAddr_AxisZ: 1001, iSlaveAddr_AxisS: 1003, IxTorqueOverload: IxTorqueOverload_St1, T_Station_Parameter: T_NovRam.T_Parameter.T_StationWork[gciStationSt1], T_Station_Work: TStation_Work_St1, IuiActualTorqueAxisZ: IuiActualTorqueAxisZ_St1, IwInputState_Z_Axis: wState_Z_Axis_St1, IuiActualTorqueAxisS: IuiActualTorqueAxisS_St1, IwInputState_S1_Axis: IwInputState_S1_Axis_St1, IwInputState_S2_Axis: IwInputState_S2_Axis_St1, IwInputState_S3_Axis: IwInputState_S3_Axis_St1, stZRefIn: stZRefIn_St1, stZRefOut: stZRefOut_St1, stZDriveState: stZDriveState_St1, stSRefIn: stSRefIn_St1, stSRefOut: stSRefOut_St1, stS2RefIn: stS2RefIn_St1, stS2RefOut: stS2RefOut_St1, stS3RefIn: stS3RefIn_St1, stS3RefOut: stS3RefOut_St1, T_HDD: T_HDD, T_TwinSafe_Ctrle_Z_Axis: T_TwinSafe_Ctrle_Z_Axis_St1, T_TwinSafe_Status_Z_Axis: T_TwinSafe_Status_Z_Axis_St1, T_TwinSafe_Ctrle_S2_Axis: T_TwinSafe_Ctrle_S2_Axis_St1, T_TwinSafe_Status_S2_Axis: T_TwinSafe_Status_S2_Axis_St1, T_TwinSafe_Ctrle_S3_Axis: T_TwinSafe_Ctrle_S3_Axis_St1, T_TwinSafe_Status_S3_Axis: T_TwinSafe_Status_S3_Axis_St1, stBubblerDataIN: stBubblerDataINSt1, stBubblerDataOUT: stBubblerDataOUTSt1, stFeedpumpINData: stFeedpumpINDataSt1, stFeedpumpOUTData: stFeedpumpOUTDataSt1, xActiveStation => xActiveStationWork_St1, QiAToolDeflection_SM => QiAToolDeflection_SM_St1, QiAToolTorqueHC_SM => QiAToolTorqueHC_SM_St1, QiAToolTorqueOverload_SM => QiAToolTorqueOverload_SM_St1, QxCylBrakeReleaseZAxis_Open => QxCylBrakeReleaseZAxis_Open_St1, QxCylBrakeReleaseZAxis_Close => QxCylBrakeReleaseZAxis_Close_St1, QxCylWorkpieceClamp_Close => QxCylWorkpieceClamp_St1, QxAirTable => QxAirTable, QxVacuumTable => QxVacuumTable, QxMeasRangeTorqueSensor => QxMeasRangeTorqueSensor_St1, QxControlTorqueSensor => QxControlTorqueSensor_St1) => xActiveHWWork_St1
NETWORK 5
	NOT TStation_Work_St1.TControl.xActiveHardware => >>ResetOutput_WORK
NETWORK 6
	TRUE => <RETURN>
NETWORK 7 ResetOutput_WORK:
	FALSE => QxCylBrakeReleaseZAxis_Open_St1, QxCylBrakeReleaseZAxis_Close_St1, QxCylWorkpieceClamp_St1, QxAirTable, QxVacuumTable, QxMeasRangeTorqueSensor_St1, QxControlTorqueSensor_St1
NETWORK 8
	0 => QiAToolDeflection_SM_St1, QiAToolTorqueHC_SM_St1, QiAToolTorqueOverload_SM_St1
_END_FBD_
(* the same logic as Structured Text *)
(* Network 1 *)
xStationPowerON_St1 := gT_SafetyStatus.xEnergyONNormalMode OR gT_SafetyStatus.xEnergyONSetupModeASt1 OR gT_SafetyStatus.xEnergyONSetupModeBSt1;
(* Network 2 *)
gudiTorqueOverloadCounterValueSt1 := IudiTorqueOverloadCounterValue_St1;
(* Network 3 *)
wState_Z_Axis_St1 := SEL(gxHardwareOFF OR gxAxisOFF, IwInputState_Z_Axis_St1, 24);
(* Network 4 *)
FBHWStationWork_St1(iStationNr := 1, xStationPowerON := xStationPowerON_St1, IxToolDeflection := IxToolDeflection_St1, IiAToolTorque := IiAToolTorque_St1, IiAToolTorque2 := IiAToolTorque2_St1, IxBrakeReleaseZAxis := IxBrakeReleaseZ1Axis_St1, IxUpperToolGuide_WorkpieceClamped := IxUpperToolGuide_WorkpieceClamped_St1, IbTooSpindleActive := T_ExchgParam.bToolSpindleActive, iSlaveAddr_AxisZ := 1001, iSlaveAddr_AxisS := 1003, IxTorqueOverload := IxTorqueOverload_St1, T_Station_Parameter := T_NovRam.T_Parameter.T_StationWork[gciStationSt1], T_Station_Work := TStation_Work_St1, IuiActualTorqueAxisZ := IuiActualTorqueAxisZ_St1, IwInputState_Z_Axis := wState_Z_Axis_St1, IuiActualTorqueAxisS := IuiActualTorqueAxisS_St1, IwInputState_S1_Axis := IwInputState_S1_Axis_St1, IwInputState_S2_Axis := IwInputState_S2_Axis_St1, IwInputState_S3_Axis := IwInputState_S3_Axis_St1, stZRefIn := stZRefIn_St1, stZRefOut := stZRefOut_St1, stZDriveState := stZDriveState_St1, stSRefIn := stSRefIn_St1, stSRefOut := stSRefOut_St1, stS2RefIn := stS2RefIn_St1, stS2RefOut := stS2RefOut_St1, stS3RefIn := stS3RefIn_St1, stS3RefOut := stS3RefOut_St1, T_HDD := T_HDD, T_TwinSafe_Ctrle_Z_Axis := T_TwinSafe_Ctrle_Z_Axis_St1, T_TwinSafe_Status_Z_Axis := T_TwinSafe_Status_Z_Axis_St1, T_TwinSafe_Ctrle_S2_Axis := T_TwinSafe_Ctrle_S2_Axis_St1, T_TwinSafe_Status_S2_Axis := T_TwinSafe_Status_S2_Axis_St1, T_TwinSafe_Ctrle_S3_Axis := T_TwinSafe_Ctrle_S3_Axis_St1, T_TwinSafe_Status_S3_Axis := T_TwinSafe_Status_S3_Axis_St1, stBubblerDataIN := stBubblerDataINSt1, stBubblerDataOUT := stBubblerDataOUTSt1, stFeedpumpINData := stFeedpumpINDataSt1, stFeedpumpOUTData := stFeedpumpOUTDataSt1);
xActiveStationWork_St1 := FBHWStationWork_St1.xActiveStation;
QiAToolDeflection_SM_St1 := FBHWStationWork_St1.QiAToolDeflection_SM;
QiAToolTorqueHC_SM_St1 := FBHWStationWork_St1.QiAToolTorqueHC_SM;
QiAToolTorqueOverload_SM_St1 := FBHWStationWork_St1.QiAToolTorqueOverload_SM;
QxCylBrakeReleaseZAxis_Open_St1 := FBHWStationWork_St1.QxCylBrakeReleaseZAxis_Open;
QxCylBrakeReleaseZAxis_Close_St1 := FBHWStationWork_St1.QxCylBrakeReleaseZAxis_Close;
QxCylWorkpieceClamp_St1 := FBHWStationWork_St1.QxCylWorkpieceClamp_Close;
QxAirTable := FBHWStationWork_St1.QxAirTable;
QxVacuumTable := FBHWStationWork_St1.QxVacuumTable;
QxMeasRangeTorqueSensor_St1 := FBHWStationWork_St1.QxMeasRangeTorqueSensor;
QxControlTorqueSensor_St1 := FBHWStationWork_St1.QxControlTorqueSensor;
xActiveHWWork_St1 := FBHWStationWork_St1.xActiveHWStation;
(* Network 5 *)
IF NOT TStation_Work_St1.TControl.xActiveHardware THEN JMP ResetOutput_WORK; END_IF;
(* Network 6 *)
RETURN;
(* Network 7 *)
ResetOutput_WORK:
QxCylBrakeReleaseZAxis_Open_St1 := FALSE;
QxCylBrakeReleaseZAxis_Close_St1 := FALSE;
QxCylWorkpieceClamp_St1 := FALSE;
QxAirTable := FALSE;
QxVacuumTable := FALSE;
QxMeasRangeTorqueSensor_St1 := FALSE;
QxControlTorqueSensor_St1 := FALSE;
(* Network 8 *)
QiAToolDeflection_SM_St1 := 0;
QiAToolTorqueHC_SM_St1 := 0;
QiAToolTorqueOverload_SM_St1 := 0;
END_PROGRAM

(* POU PRG_LAYER2_HARDWARE/PRG_HW_GENERAL, FBD *)
PROGRAM PRG_HW_GENERAL
VAR
(* CPU *)
	(* function bloc *)
	(* IO connection *)
(* Fieldbus *)
	(* function bloc *)
	(* IO connection *)
	FBHWHdd: FBHW_HDD;
	fbNovRam: FBHW_NOVRAM;
	fbProfileFile:FB_PROFILE_FILE;
	FBPassword:FB_PASSWORD;
	FBProcessData_St1: FB_PROCESSDATA;
	fbGetUPSStatus: FB_GetUPSStatus;
	xValid: BOOL;
	xError: BOOL;
	udiErrorNr: UDINT;
	FBControlLamp: FB_ControlLamp;
	FBHW_MachineLamp: FBHW_CYL_STANDARD;
END_VAR
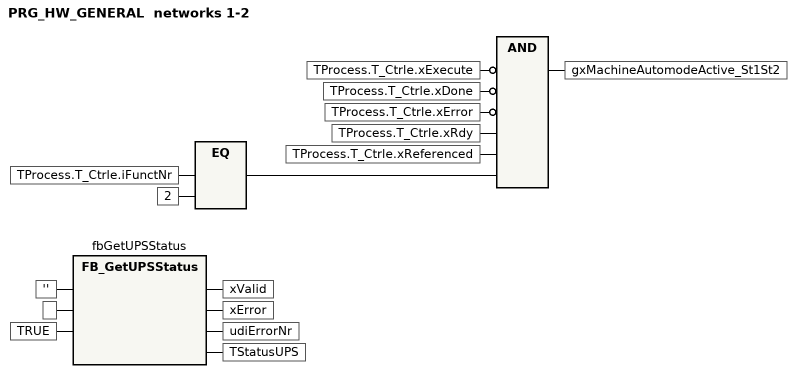
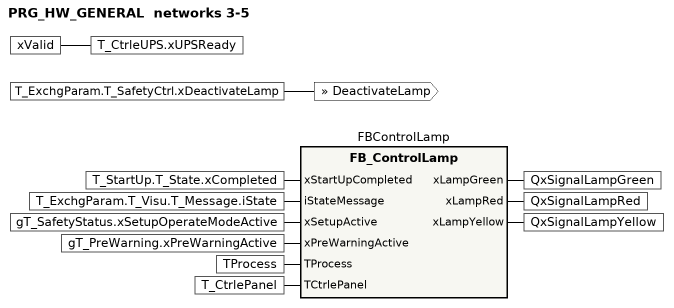
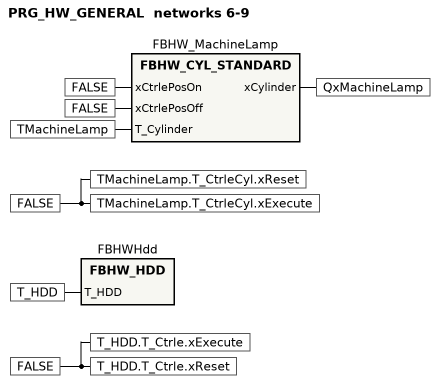
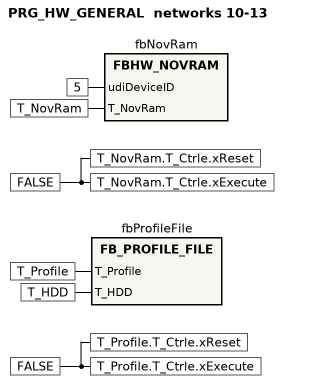
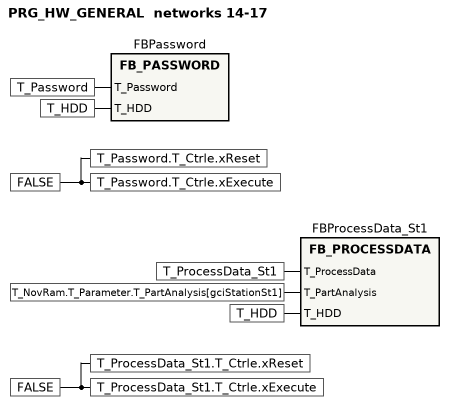
_FBD_ (* Function Block Diagram *)
NETWORK 1
	AND(NOT TProcess.T_Ctrle.xExecute, NOT TProcess.T_Ctrle.xDone, NOT TProcess.T_Ctrle.xError, TProcess.T_Ctrle.xRdy, TProcess.T_Ctrle.xReferenced, EQ(TProcess.T_Ctrle.iFunctNr, 2)) => gxMachineAutomodeActive_St1St2
NETWORK 2
	fbGetUPSStatus:FB_GetUPSStatus('', , TRUE, out 2 => xError, out 3 => udiErrorNr, out 4 => TStatusUPS) => xValid
NETWORK 3
	xValid => T_CtrleUPS.xUPSReady
NETWORK 4
	T_ExchgParam.T_SafetyCtrl.xDeactivateLamp => >>DeactivateLamp
NETWORK 5
	FBControlLamp:FB_ControlLamp(xStartUpCompleted: T_StartUp.T_State.xCompleted, iStateMessage: T_ExchgParam.T_Visu.T_Message.iState, xSetupActive: gT_SafetyStatus.xSetupOperateModeActive, xPreWarningActive: gT_PreWarning.xPreWarningActive, TProcess: TProcess, TCtrlePanel: T_CtrlePanel, xLampRed => QxSignalLampRed, xLampYellow => QxSignalLampYellow) => QxSignalLampGreen
NETWORK 6
	FBHW_MachineLamp:FBHW_CYL_STANDARD(xCtrlePosOn: FALSE, xCtrlePosOff: FALSE, T_Cylinder: TMachineLamp) => QxMachineLamp
NETWORK 7 DeactivateLamp:
	FALSE => TMachineLamp.T_CtrleCyl.xReset, TMachineLamp.T_CtrleCyl.xExecute
NETWORK 8
	FBHWHdd:FBHW_HDD(T_HDD: T_HDD)
NETWORK 9
	FALSE => T_HDD.T_Ctrle.xExecute, T_HDD.T_Ctrle.xReset
NETWORK 10
	fbNovRam:FBHW_NOVRAM(udiDeviceID: 5, T_NovRam: T_NovRam)
NETWORK 11
	FALSE => T_NovRam.T_Ctrle.xReset, T_NovRam.T_Ctrle.xExecute
NETWORK 12
	fbProfileFile:FB_PROFILE_FILE(T_Profile: T_Profile, T_HDD: T_HDD)
NETWORK 13
	FALSE => T_Profile.T_Ctrle.xReset, T_Profile.T_Ctrle.xExecute
NETWORK 14
	FBPassword:FB_PASSWORD(T_Password: T_Password, T_HDD: T_HDD)
NETWORK 15
	FALSE => T_Password.T_Ctrle.xReset, T_Password.T_Ctrle.xExecute
NETWORK 16
	FBProcessData_St1:FB_PROCESSDATA(T_ProcessData: T_ProcessData_St1, T_PartAnalysis: T_NovRam.T_Parameter.T_PartAnalysis[gciStationSt1], T_HDD: T_HDD)
NETWORK 17
	FALSE => T_ProcessData_St1.T_Ctrle.xReset, T_ProcessData_St1.T_Ctrle.xExecute
_END_FBD_
END_PROGRAM

(* POU FB_HARDWARE/FBHW_HDD, ST *)
FUNCTION_BLOCK FBHW_HDD
VAR_INPUT
END_VAR
VAR_OUTPUT
END_VAR
VAR_IN_OUT
	T_HDD:ST_HDD;
END_VAR
VAR
(* variable *)
	xConfirmResetFB: BOOL;
	i:INT;
	dwOpenFileMod:DWORD;
	udiHdleFile:UINT;
	xFileOpen: BOOL;
	xFileClose:BOOL;
	xFileRead:BOOL;
	xFileAppendWrite:BOOL;
	xFileCreate:BOOL;
	xFileBiggerAsMaxLine:BOOL;
	xFileDelete: BOOL;
	xRenameFile:BOOL;
(* function bloc *)
	fbFileOpen:FB_FileOpen;
	fbFileWrite:FB_FileWrite;
	fbFileClose:FB_FileClose;
	fbFileGets:FB_FileGets;
	fbFilePuts:FB_FilePuts;
	fbFileDelete:FB_FileDelete;
	fbRenameFile:FB_FileRename;
	fbCreateDir:FB_CreateDir;
	fbRemoveDir:FB_RemoveDir;
(* Trigger *)
	RisingEdgeExecute:R_TRIG;
	RisingEdgeReset:R_TRIG;
	xCreateDirectory: BOOL;
	xRemoveDirectory: BOOL;
	xFileWrite: BOOL;
	ii: INT;
	iCalcLenght: INT;
	jj: INT;
	xFileReadComplete: BOOL;
	fbFileRead: FB_FileRead;
	xFileRead1Line: BOOL;
	xConvertData: BOOL;
	iStepConvertData: INT;
	iStartPoint: INT;
	iStopPoint: INT;
	iStepLength: INT;
	diStepCounter: DINT;
	asCopyString: ARRAY [1..255] OF STRING(255);
	xFirstTime: BOOL;
END_VAR
(* waiting for reset *)
	RisingEdgeReset(CLK:=T_HDD.T_Ctrle.xReset);
	IF RisingEdgeReset.Q THEN
	(* init. function bloc *)
		fbFileOpen(bExecute:=FALSE);
		fbFileClose(bExecute:=FALSE);
		fbFileWrite(bExecute:=FALSE);
		fbFileGets(bExecute:=FALSE);
		fbFilePuts(bExecute:=FALSE);
		fbFileDelete(bExecute:=FALSE);
		fbRenameFile(bExecute:=FALSE);
	(* init. variable *)
		dwOpenFileMod:=0;
		udiHdleFile:=0;
		xFileOpen:=FALSE;
		xFileClose:=FALSE;
		xFileRead:=FALSE;
		xFileRead1Line:=FALSE;
		xFileAppendWrite:=FALSE;
		xFileCreate:=FALSE;
		xFileWrite:=FALSE;
		xFileReadComplete:=FALSE;
		xFileBiggerAsMaxLine:=FALSE;
		xFileDelete:=FALSE;
		xRenameFile:=FALSE;
	(* init. structure *)
		T_HDD.T_Ctrle.xDone:=FALSE;
		T_HDD.T_Ctrle.xErr:=FALSE;
		T_HDD.T_Ctrle.udiErrorID:=0;
		T_HDD.T_Ctrle.iFunction:=0;
		T_HDD.T_File.sPathAndFileName:='';
		T_HDD.T_File.sOldPathAndFileName:='';
		T_HDD.T_Ctrle.tTimeOut:=T#2s;
		T_HDD.T_Ctrle.xLocked:=FALSE;
		IF NOT(xFirstTime) THEN
			xFirstTime:=TRUE;
			FOR ii:= 1 TO 255 DO
				asCopyString[ii]:='';
			END_FOR;
			FOR ii:= 1 TO 255 DO
				FOR jj:=1 TO ii DO
					asCopyString[ii]:=CONCAT(asCopyString[ii],' ');
				END_FOR;
				IF (ii = 250) THEN
					iCalcLenght:=LEN(asCopyString[ii]);
				END_IF;
			END_FOR;
		END_IF;
		(* set flag done *)
		xConfirmResetFB:=TRUE;
		(* exit function *)
		RETURN;
	ELSE
		IF xConfirmResetFB THEN
		(* confirm reset FB *)
			T_HDD.T_Ctrle.xDone:=TRUE;
			T_HDD.T_Ctrle.xErr:=FALSE;
			T_HDD.T_Ctrle.udiErrorID:=0;
			T_HDD.T_Ctrle.xLocked:=FALSE;
			(* init. variable *)
			xConfirmResetFB:=FALSE;
		END_IF
	END_IF

(* waiting for execute *)
	RisingEdgeExecute(CLK:=T_HDD.T_Ctrle.xExecute);
	IF RisingEdgeExecute.Q THEN
		CASE T_HDD.T_Ctrle.iFunction OF
		(* Read file *)
		1:	(* activ file open *)
			xFileOpen:=TRUE;
			dwOpenFileMod:=FOPEN_MODEREAD OR FOPEN_MODEPLUS OR FOPEN_MODETEXT;
		(* Write file *)
		2:	(* activ file open *)
			xFileOpen:=TRUE;
			dwOpenFileMod:=FOPEN_MODEWRITE OR FOPEN_MODEPLUS OR FOPEN_MODETEXT;
		(* overwrite file *)
		3:	(* activ file open *)
			xFileOpen:=TRUE;
			dwOpenFileMod:=FOPEN_MODEAPPEND OR FOPEN_MODEPLUS OR FOPEN_MODETEXT;
		(* file exists *)
		4:	(* activ file open *)
			xFileOpen:=TRUE;
			dwOpenFileMod:=FOPEN_MODEREAD OR FOPEN_MODEPLUS OR FOPEN_MODETEXT;
		(* delete file *)
		5:	xFileDelete:=TRUE;
		(* rename file *)
		6:	xRenameFile:=TRUE;
		(* create directory *)
		7:	xCreateDirectory:=TRUE;
		(* remove directory *)
		8:	xRemoveDirectory:=TRUE;
		(* Read file complete *)
		9:	(* activ file open *)
			xFileOpen:=TRUE;
			dwOpenFileMod:=FOPEN_MODEREAD OR FOPEN_MODEPLUS OR FOPEN_MODETEXT;
		(* Write file complete *)
		10:	(* activ file open *)
			xFileOpen:=TRUE;
			dwOpenFileMod:=FOPEN_MODEWRITE OR FOPEN_MODETEXT ;
		(* Read File only 1 line *)
		11:	(* activ file open *)
			xFileOpen:=TRUE;
			dwOpenFileMod:=FOPEN_MODEREAD OR FOPEN_MODEPLUS OR FOPEN_MODETEXT;
		ELSE
		(* function not implemented *)
			 T_HDD.T_Ctrle.xDone:=FALSE;
			 T_HDD.T_Ctrle.xErr:=TRUE;
			 T_HDD.T_Ctrle.udiErrorID:=16#F000;
			 T_HDD.T_Ctrle.xLocked:=FALSE;
			 (* exit FB *)
			 RETURN;
		END_CASE
		(* Init. variable *)
		T_HDD.T_Ctrle.xDone:=FALSE;
		T_HDD.T_Ctrle.xErr:=FALSE;
		T_HDD.T_Ctrle.udiErrorID:=16#0;
		xFileBiggerAsMaxLine:=FALSE;
		(* init. variable*)
		i:=1;
		RETURN;
	END_IF

(* Open file *)
	IF xFileOpen THEN
		fbFileOpen(	sNetId:=T_HDD.T_Config.sNetId,
					sPathName:=T_HDD.T_File.sPathAndFileName,
					nMode:=dwOpenFileMod,
					ePath := PATH_GENERIC,
					bExecute:=TRUE,
					tTimeout:=T#2s);
		IF NOT(fbFileOpen.bBusy) OR fbFileOpen.bError THEN
			IF NOT(fbFileOpen.bError) THEN
				CASE T_HDD.T_Ctrle.iFunction OF
				1:	xFileRead:=TRUE;
				2:	xFileCreate:=TRUE;
				3: 	xFileAppendWrite:=TRUE;
				4:	xFileClose:=TRUE;
				9:	xFileReadComplete:=TRUE;
				10:	xFileWrite:=TRUE;
(*
					FOR ii:=1 TO csiMaxFileLine DO
						iCalcLenght:=LEN(T_HDD.T_Data.sData[ii]);
						iMaxChar:=SIZEOF(T_HDD.T_Data.sData[ii]);
						iCheckElement:=(iMaxChar - 2) - iCalcLenght;
						T_HDD.T_Data.sData[ii]:=CONCAT(T_HDD.T_Data.sData[ii],asCopyString[iCheckElement]);
						iCalcLenght:=LEN(T_HDD.T_Data.sData[ii]);
						T_HDD.T_Data.sData[ii]:=CONCAT(T_HDD.T_Data.sData[ii],'$L');
						iCalcLenght:=LEN(T_HDD.T_Data.sData[ii]);
						IF (ii = 250) THEN
							iCalcLenght:=LEN(T_HDD.T_Data.sData[ii]);
						END_IF;
					END_FOR;
*)
				11:	xFileRead1Line:=TRUE;
				END_CASE
				(* Handle file *)
				udiHdleFile:=fbFileOpen.hFile;
			ELSE
				udiHdleFile:=0;
				 T_HDD.T_Ctrle.xDone:= FALSE;
				 T_HDD.T_Ctrle.xErr:=fbFileOpen.bError;
				 T_HDD.T_Ctrle.udiErrorID:=fbFileOpen.nErrId;
				 T_HDD.T_Ctrle.xLocked:=FALSE;
			END_IF
			(* set flag xfileopen off *)
			xFileOpen:=FALSE;
		END_IF
	ELSE fbFileOpen(bExecute:=FALSE); END_IF

(* Read file *)
	IF xFileRead OR xFileRead1Line THEN
		fbFileGets(	sNetId:=T_HDD.T_Config.sNetId,
					hFile:=udiHdleFile,
					bExecute:=TRUE,
					tTimeOut:=T_HDD.T_Ctrle.tTimeOut);
		IF NOT(fbFileGets.bBusy) OR fbFileGets.bError THEN
			T_HDD.T_Data.sData[i]:=fbFileGets.sLine;
			(* check eof or error *)
			IF fbFileGets.bEOF OR fbFileGets.bError OR i = csiMaxFileLine OR xFileRead1Line THEN
				 (* set flag xFileRead off *)
				 xFileRead:=FALSE;
				xFileRead1Line:=FALSE;
				 (* activ closing file *)
				 xFileClose:=TRUE;
				 (* activ variable file bigger as structure *)
				 IF i = csiMaxFileLine THEN xFileBiggerAsMaxLine:=TRUE; END_IF
			ELSE
			(* read next line *)
				fbFileGets(bExecute:=FALSE);
				i:=i+1;
			END_IF
		END_IF
	ELSE fbFileGets(bExecute:=FALSE); END_IF

(* Write at the end of file or create file *)
	IF xFileAppendWrite OR xFileCreate THEN
		fbFilePuts(	sNetId:=T_HDD.T_Config.sNetId,
					hFile:=udiHdleFile,
					sLine:=CONCAT(T_HDD.T_Data.sData[i],'$L'),
					bExecute:=TRUE,
					tTimeOut:=T_HDD.T_Ctrle.tTimeOut);
		IF NOT(fbFilePuts.bBusy) OR fbFilePuts.bError THEN
			IF T_HDD.T_Data.sData[i+1] = '' THEN
				 (* set flag xFileCreate or xFileAppendWrite off *)
				xFileAppendWrite:=FALSE;
				xFileCreate:=FALSE;
				 (* activ closing file *)
				 xFileClose:=TRUE;
			ELSE
			(* Init. FB *)
				 fbFilePuts(bExecute:=FALSE);
				 (* next line *)
				i:=i+1;
			END_IF
		END_IF
	ELSE IF NOT(xFileAppendWrite) AND NOT(xFileCreate) THEN fbFilePuts(bExecute:=FALSE); END_IF
	END_IF

(* Read the hole file file *)
	IF xFileReadComplete THEN
		fbFileRead(	sNetId:= T_HDD.T_Config.sNetId,
					hFile:= udiHdleFile,
					pReadBuff:=ADR(T_HDD.T_Data.sData),
					cbReadLen:=SIZEOF(T_HDD.T_Data.sData),
					bExecute:= TRUE,
					tTimeout:=T_HDD.T_Ctrle.tTimeOut);
		IF NOT(fbFileRead.bBusy) OR fbFileRead.bError THEN
			fbFileRead(bExecute:=FALSE);
			xFileReadComplete:=FALSE;
			xConvertData:=TRUE;
			iStepConvertData:=1;
		END_IF
	ELSE fbFileRead(bExecute:=FALSE); END_IF
	IF xConvertData THEN
		CASE iStepConvertData OF
		1:	iStartPoint:=1;
			iStepLength:=csiMaxFileLine / 24;
			iStopPoint:=iStartPoint + iStepLength;
			diStepCounter:=0;
			FOR ii:=iStartPoint TO iStopPoint DO
				diStepCounter:=diStepCounter + 1;
				T_HDD.T_Data.sData[ii]:=sFctDeleteChar(T_HDD.T_Data.sData[ii],' ');
				T_HDD.T_Data.sData[ii]:=sFctDeleteChar(T_HDD.T_Data.sData[ii],'$N');
				T_HDD.T_Data.sData[ii]:=sFctDeleteChar(T_HDD.T_Data.sData[ii],'$L');
			END_FOR;
			iStepConvertData:=iStepConvertData + 1;
		2:	iStartPoint:=iStopPoint;
			iStopPoint:=iStartPoint + iStepLength;
			IF (iStartPoint > csiMaxFileLine) THEN iStartPoint:=csiMaxFileLine; END_IF;
			IF (iStopPoint > csiMaxFileLine) THEN iStopPoint:=csiMaxFileLine; END_IF;
			FOR ii:=iStartPoint TO iStopPoint DO
				diStepCounter:=diStepCounter + 1;
				T_HDD.T_Data.sData[ii]:=sFctDeleteChar(T_HDD.T_Data.sData[ii],' ');
				T_HDD.T_Data.sData[ii]:=sFctDeleteChar(T_HDD.T_Data.sData[ii],'$N');
				T_HDD.T_Data.sData[ii]:=sFctDeleteChar(T_HDD.T_Data.sData[ii],'$L');
			END_FOR;
			iStepConvertData:=iStepConvertData + 1;
		3:	IF (iStopPoint >= csiMaxFileLine) THEN
				iStepConvertData:=iStepConvertData + 1;
			ELSE
				iStepConvertData:=2;
			END_IF;
		4:	(* activ closing file *)
			xConvertData:=FALSE;
			iStepConvertData:=1;
			 xFileClose:=TRUE;
		END_CASE;
	END_IF;

(* Write at the end of file or create file *)
	IF xFileWrite THEN
		fbFileWrite(	sNetId:= T_HDD.T_Config.sNetId,
					hFile:= udiHdleFile,
					pWriteBuff:= ADR(T_HDD.T_Data.sData),
					cbWriteLen:= SIZEOF(T_HDD.T_Data.sData),
					bExecute:= TRUE,
					tTimeout:=T_HDD.T_Ctrle.tTimeOut);
		IF NOT(fbFileWrite.bBusy) OR fbFileWrite.bError THEN
			fbFileWrite(bExecute:=FALSE);
			xFileWrite:=FALSE;
			(* activ closing file *)
			 xFileClose:=TRUE;
		END_IF
	ELSE fbFileWrite(bExecute:=FALSE); END_IF

(* Close file *)
	IF xFileClose THEN
		fbFileClose(	sNetId:=T_HDD.T_Config.sNetId,
					hFile:=udiHdleFile,
					bExecute:=TRUE,
					tTimeout:=T#2s);
		IF NOT(fbFileClose.bBusy) OR fbFileClose.bError THEN
			 T_HDD.T_Ctrle.xDone:= NOT(fbFileClose.bBusy);
			 T_HDD.T_Ctrle.xErr:=fbFileClose.bError;
			 T_HDD.T_Ctrle.udiErrorID:=fbFileClose.nErrId;
			 udiHdleFile:=0;
			(* check if file bigger as maximum reading line *)
			IF xFileBiggerAsMaxLine THEN
				T_HDD.T_Ctrle.xErr:=TRUE;
				T_HDD.T_Ctrle.udiErrorID:=16#F501;
			END_IF
			 (* set flag xFileClose off *)
			 xFileClose:=FALSE;
		END_IF
	ELSE fbFileClose(bExecute:=FALSE); END_IF

(* Delete file *)
	IF xFileDelete THEN
		fbFileDelete(	sNetId:=T_HDD.T_Config.sNetId,
					sPathName:=T_HDD.T_File.sPathAndFileName,
					bExecute:=TRUE,
					tTimeout:=T#2s);
		IF NOT(fbFileDelete.bBusy) OR fbFileDelete.bError THEN
			 T_HDD.T_Ctrle.xDone:= NOT(fbFileDelete.bBusy);
			 T_HDD.T_Ctrle.xErr:=fbFileDelete.bError;
			 T_HDD.T_Ctrle.udiErrorID:=fbFileDelete.nErrId;
			 (* set flag xFileDelete off *)
			 xFileDelete:=FALSE;
		END_IF
	ELSE fbFileDelete(bExecute:=FALSE); END_IF

(* rename file *)
	IF xRenameFile THEN
		fbRenameFile(	sNetId:=T_HDD.T_Config.sNetId,
						sOldName:=T_HDD.T_File.sOldPathAndFileName,
						sNewName:=T_HDD.T_File.sPathAndFileName,
						ePath:=PATH_GENERIC,
						bExecute:=TRUE,
						tTimeout:=T#2s);
		IF NOT(fbRenameFile.bBusy) OR fbRenameFile.bError THEN
			 T_HDD.T_Ctrle.xDone:= NOT(fbRenameFile.bBusy);
			 T_HDD.T_Ctrle.xErr:=fbRenameFile.bError;
			 T_HDD.T_Ctrle.udiErrorID:=fbRenameFile.nErrId;
			 (* set flag xFileDelete off *)
			 xRenameFile:=FALSE;
		END_IF
	ELSE fbRenameFile(bExecute:=FALSE); END_IF

(* create directory *)
	IF xCreateDirectory THEN
		fbCreateDir(	sNetId:= T_HDD.T_Config.sNetId,
					sPathName:= T_HDD.T_File.sDirectoryPath,
					ePath:= PATH_GENERIC,
					bExecute:= TRUE,
					tTimeout:= T#2s);
		IF NOT(fbCreateDir.bBusy) OR fbCreateDir.bError THEN
			 T_HDD.T_Ctrle.xDone:= NOT(fbCreateDir.bBusy);
			 T_HDD.T_Ctrle.xErr:=fbCreateDir.bError;
			 T_HDD.T_Ctrle.udiErrorID:=fbCreateDir.nErrId;
			 (* set flag xFileDelete off *)
			 xCreateDirectory:=FALSE;
		END_IF;
	ELSE fbCreateDir(	sNetId:= T_HDD.T_Config.sNetId,
					sPathName:= T_HDD.T_File.sDirectoryPath,
					ePath:= PATH_GENERIC,
					bExecute:= FALSE,
					tTimeout:= T#2s);
	END_IF;

(* remove directory *)
	IF xRemoveDirectory THEN
		(* Verzeichnis kann nur gelöscht werden falls es keine Dateien enthält, anderenfalls wird es nicht gelöscht und diese Funktion setzt einen Fehler *)
		fbRemoveDir(	sNetId:= T_HDD.T_Config.sNetId,
						sPathName:= T_HDD.T_File.sDirectoryPath,
						ePath:= PATH_GENERIC,
						bExecute:= TRUE,
						tTimeout:= T#2s);
		IF NOT(fbRemoveDir.bBusy) OR fbRemoveDir.bError THEN
			 T_HDD.T_Ctrle.xDone:= NOT(fbRemoveDir.bBusy);
			 T_HDD.T_Ctrle.xErr:=fbRemoveDir.bError;
			 T_HDD.T_Ctrle.udiErrorID:=fbRemoveDir.nErrId;
			 (* set flag xFileDelete off *)
			 xRemoveDirectory:=FALSE;
		END_IF;
	ELSE fbRemoveDir(	sNetId:= T_HDD.T_Config.sNetId,
						sPathName:= T_HDD.T_File.sDirectoryPath,
						ePath:= PATH_GENERIC,
						bExecute:= FALSE,
						tTimeout:= T#2s);
	END_IF;
END_FUNCTION_BLOCK

(* POU GENERAL/sFctDeleteChar, ST *)
FUNCTION sFctDeleteChar : STRING(255)
VAR_INPUT
	sString:STRING(255);
	sChar:STRING(1);
END_VAR
VAR
	sCopyString: STRING(255);
	iFindChar: INT;
END_VAR
sFctDeleteChar:='';
sCopyString:=sString;
WHILE (FIND(sCopyString,sChar) <> 0) DO
	iFindChar:=FIND(sCopyString,sChar);
	sCopyString:=DELETE(sCopyString,1,iFindChar);
END_WHILE;
sFctDeleteChar:=sCopyString;
END_FUNCTION

(* POU FB_HARDWARE/FBHW_NOVRAM, ST *)
FUNCTION_BLOCK FBHW_NOVRAM
VAR_INPUT
	udiDeviceID:UDINT;
END_VAR
VAR_IN_OUT
	T_NovRam:ST_NOVRAM;
END_VAR
VAR_OUTPUT
END_VAR
VAR
(* function bloc *)
	fbNovRamReadWrite:FB_NovRamReadWrite;
(* trigger *)
	RisingEdgeResetFB:R_TRIG;
	RisingEdgeExecute:R_TRIG;
(* variable *)
	xRead:BOOL:=FALSE;
	xWrite:BOOL:=FALSE;
	xConfirmResetFB: BOOL;
END_VAR
(* reset *)
	RisingEdgeResetFB(CLK:=T_NovRam.T_Ctrle.xReset);
	IF RisingEdgeResetFB.Q THEN
	(* init. variable *)
		xRead:=FALSE;
		xWrite:=FALSE;
	(* activ confirmation reset *)
		xConfirmResetFB:=TRUE;
	(* Exit FB *)
		RETURN;
	ELSE
		IF xConfirmResetFB THEN
		(* confirm reset FB *)
			T_NovRam.T_Ctrle.xDone:=TRUE;
			T_NovRam.T_Ctrle.xErr:=FALSE;
			T_NovRam.T_Ctrle.udiErrorID:=16#0;
		(* reset variable *)
			xConfirmResetFB:=FALSE;
		END_IF
	END_IF

(* execute *)
	RisingEdgeExecute(CLK:=T_NovRam.T_Ctrle.xExecute);
	IF RisingEdgeExecute.Q THEN
		(* init. capacity and pointer *)
		T_NovRam.T_Ctrle.udipSrcAddr:=ADR(T_NovRam.T_Parameter);
		T_NovRam.T_Ctrle.udiSrcLen:=SIZEOF(T_NovRam.T_Parameter);
		T_NovRam.T_Ctrle.udipDestAddr:=ADR(T_NovRam.T_Parameter);
		T_NovRam.T_Ctrle.udiDestLen:=SIZEOF(T_NovRam.T_Parameter);
		CASE T_NovRam.T_Ctrle.iFunction OF
		(* Read *)
		1:	xRead:=TRUE;
		(* Write *)
		2:	xWrite:=TRUE;
		ELSE
		(* function not implemented *)
			T_NovRam.T_Ctrle.xDone:=FALSE;
			T_NovRam.T_Ctrle.xErr:=TRUE;
			T_NovRam.T_Ctrle.udiErrorID:=16#F000;
			(* Exit FB *)
			RETURN;
		END_CASE
		(* Init. variable *)
		T_NovRam.T_Ctrle.xDone:=FALSE;
		T_NovRam.T_Ctrle.xErr:=FALSE;
		T_NovRam.T_Ctrle.udiErrorID:=0;
	(* Exit FB *)
		RETURN;
	END_IF

(* wait for read/write *)
	IF xRead OR xWrite THEN
		IF NOT(gxHardwareOFF) THEN
			fbNovRamReadWrite(	nDevId:=udiDeviceID,
								bRead:=xRead,
								bWrite:=xWrite,
								cbSrcLen:=T_NovRam.T_Ctrle.udiSrcLen,
								cbDestLen:=T_NovRam.T_Ctrle.udiDestLen,
								pSrcAddr:=T_NovRam.T_Ctrle.udipSrcAddr,
								pDestAddr:=T_NovRam.T_Ctrle.udipDestAddr,
								tTimeOut:=T_NovRam.T_Ctrle.tTimeOut);
			IF NOT(fbNovRamReadWrite.bBusy) OR fbNovRamReadWrite.bError THEN
				IF fbNovRamReadWrite.bError THEN
				(* set error *)
					T_NovRam.T_Ctrle.xDone:=FALSE;
					T_NovRam.T_Ctrle.xErr:=TRUE;
					T_NovRam.T_Ctrle.udiErrorID:=fbNovRamReadWrite.nErrId;
				ELSE
				(* confirm execution *)
					IF xRead THEN
						IF NOT(T_NovRam.T_Ctrle.xBlockReadFirstTime) THEN
							T_NovRam.T_Ctrle.xFirstRead:=TRUE;
						ELSE
							T_NovRam.T_Ctrle.xFirstRead:=FALSE;
						END_IF;
						T_NovRam.T_Ctrle.xBlockReadFirstTime:=FALSE;
					END_IF
					T_NovRam.T_Ctrle.xDone:=TRUE;
					T_NovRam.T_Ctrle.xErr:=FALSE;
					T_NovRam.T_Ctrle.udiErrorID:=0;
				END_IF
				(* reset variable *)
				xRead:=FALSE;
				xWrite:=FALSE;
			END_IF
		ELSE
			T_NovRam.T_Ctrle.xDone:=TRUE;
			T_NovRam.T_Ctrle.xErr:=FALSE;
			T_NovRam.T_Ctrle.udiErrorID:=0;
			(* reset variable *)
			xRead:=FALSE;
			xWrite:=FALSE;
		END_IF;
	ELSE
		fbNovRamReadWrite(	nDevId:=udiDeviceID,
							bRead:=FALSE,
							bWrite:=FALSE);
	END_IF
END_FUNCTION_BLOCK

(* POU GENERAL/PROFILE/FB_PROFILE_FILE, ST *)
FUNCTION_BLOCK FB_PROFILE_FILE
VAR_INPUT
END_VAR
VAR_OUTPUT
END_VAR
VAR_IN_OUT
	T_Profile:ST_PROFILE;
	T_HDD:ST_HDD;
END_VAR
VAR
(* Timer *)
	TimerOut:TON;
(* Trigger *)
	RisingEdgeReset:R_TRIG;
	RisingEdgeExecute:R_TRIG;
(* variable *)
	xConfirmResetFB:BOOL;
	xReadProfile:BOOL;
	xWriteProfile:BOOL;
	xReadProfileListeStation: BOOL;
	iStepFunction:INT;
	xStepFunctionDone:BOOL;
	iProfileNr:INT;
	tTimeOut: TIME;
	sDeleteData: ARRAY[1..csiMaxFileLine] OF STRING(csiMaxCharPerLine);
(* Tmp *)
	xTmp:BOOL;
	sTmp:STRING(255);
	xCheckUSBStick: BOOL;
	TimerFileLocked:TON;
	xCreateDefaultProfile: BOOL;
	T_DeleteIDProfileStation:ARRAY[1..csiMaxProfile] OF ST_PROFILE_ID;
	xDeleteProfile: BOOL;
	xRenameProfile: BOOL;
	iFindChar: INT;
	jj:INT;
	FBCopyDataFileToProfile:FB_CopyDataFileToProfile;
	sDriveName: STRING;
END_VAR
(****************************************************************************************************************************************************)
(***********                                       This Functionblock manage the profile for read and write to a file                                            ************)
(****************************************************************************************************************************************************)
IF (sDriveName = '') THEN
	sDriveName:='D:\';
END_IF;
(* waiting for reset *)
	RisingEdgeReset(CLK:=T_Profile.T_Ctrle.xReset);
	IF RisingEdgeReset.Q THEN
	(* init. structure *)
		T_Profile.T_Ctrle.xDone:=FALSE;
		T_Profile.T_Ctrle.xErr:=FALSE;
		T_Profile.T_Ctrle.udiErrorID:=0;
		T_Profile.T_Ctrle.iFunction:=0;
		(* Reset HDD if error activ *)
		IF T_HDD.T_Ctrle.xErr THEN T_HDD.T_Ctrle.xReset:=TRUE; END_IF
		(* Init. variable *)
		xReadProfile:=FALSE;
		xWriteProfile:=FALSE;
		xCheckUSBStick:=FALSE;
		xReadProfileListeStation:=FALSE;
		xCreateDefaultProfile:=FALSE;
		xDeleteProfile:=FALSE;
		xRenameProfile:=FALSE;
		(* set flag done *)
		xConfirmResetFB:=TRUE;
		(* exit function *)
		RETURN;
	ELSE
		IF xConfirmResetFB THEN
		(* confirm reset FB *)
			T_Profile.T_Ctrle.xDone:=TRUE;
			T_Profile.T_Ctrle.xErr:=FALSE;
			T_Profile.T_Ctrle.udiErrorID:=0;
			T_Profile.T_Ctrle.iFunction:=0;
			(* init. variable *)
			xConfirmResetFB:=FALSE;
		END_IF
	END_IF

TimerFileLocked(IN:=TRUE, PT:=T#10S);

(* waiting for execute *)
	RisingEdgeExecute(CLK:=T_Profile.T_Ctrle.xExecute);
	IF RisingEdgeExecute.Q THEN
		CASE T_Profile.T_Ctrle.iFunction OF
		(* read profile *)
		1:	xReadProfile:=TRUE;
			T_HDD.T_Data.sData:=sDeleteData;
			tTimeOut:=T#10s;
		(* write profile *)
		2:	xWriteProfile:=TRUE;
			tTimeOut:=T#10s;
		(* check if USB Stick exist *)
		3:	xCheckUSBStick:=TRUE;
			tTimeOut:=T#5s;
		(* read profile from File *)
		4:	xReadProfile:=TRUE;
			T_HDD.T_Data.sData:=sDeleteData;
			tTimeOut:=T#20s;
		(* write profile to File *)
		5:	xWriteProfile:=TRUE;
			tTimeOut:=T#10s;
		(* read profile liste station *)
		6:	xReadProfileListeStation:=TRUE;
			tTimeOut:=T#30s;
		(* create default profile *)
		7:	xCreateDefaultProfile:=TRUE;
			tTimeOut:=T#20s;
		(* create default profile *)
		8:	xDeleteProfile:=TRUE;
			tTimeOut:=T#20s;
		(* reanme Profil name *)
		9:	xRenameProfile:=TRUE;
			tTimeOut:=T#20s;
		ELSE
		(* function not implemented *)
			 T_Profile.T_Ctrle.xDone:=FALSE;
			 T_Profile.T_Ctrle.xErr:=TRUE;
			 T_Profile.T_Ctrle.udiErrorID:=16#F000;
			 (* exit FB *)
			 RETURN;
		END_CASE
		(* Init. variable *)
		T_Profile.T_Ctrle.xDone:=FALSE;
		T_Profile.T_Ctrle.xErr:=FALSE;
		T_Profile.T_Ctrle.udiErrorID:=16#0;
		T_HDD.T_File.cssRootPLC:=cssRootUSB;
		(* init. step *)
		iStepFunction:=1;
		xStepFunctionDone:=FALSE;
		RETURN;
	END_IF

(* Monitor time out *)
	xTmp:=	NOT T_Profile.T_Ctrle.xDone
			AND NOT T_Profile.T_Ctrle.xErr;
	TimerOut(IN:=xTmp, PT:=tTimeOut);
	IF TimerOut.Q THEN iStepFunction:=99; END_IF

(* Read or Write profile *)
	IF xReadProfile OR xWriteProfile THEN
		CASE iStepFunction OF
		(* check if HDD state *)
		(* start timeout *)
		1:	TimerFileLocked(IN:=FALSE);
			iStepFunction:=10;
		(* file name and activ read or write *)
		10:	IF T_HDD.T_Ctrle.xDone AND NOT(T_HDD.T_Ctrle.xErr) AND NOT(T_HDD.T_Ctrle.xLocked) THEN
				IF xReadProfile THEN
					sTmp:=CONCAT(sDriveName,T_Profile.T_Ctrle.sPathAndFileName);
					sTmp:=CONCAT(sTmp,'STATION');
					sTmp:=CONCAT(sTmp,UINT_TO_STRING(gciStationSt1));
					sTmp:=CONCAT(sTmp,'\');
					sTmp:=CONCAT(sTmp,INT_TO_STRING(T_Profile.T_Id.iNumber));
					sTmp:=CONCAT(sTmp,'.txt');
				(* activ read *)
					IF (T_Profile.T_Ctrle.iFunction = 1) THEN
						T_HDD.T_Ctrle.iFunction:=1;
					ELSE
						T_HDD.T_Ctrle.iFunction:=1;	(* 9 does not right function *)
					END_IF;
					T_HDD.T_Ctrle.xLocked:=TRUE;
					T_HDD.T_File.sPathAndFileName:=sTmp;
					T_HDD.T_Ctrle.xExecute:=TRUE;
					T_Profile.T_Ctrle.sProfileName:='';
					(* next step *)
					iStepFunction:=20;
					xStepFunctionDone:=FALSE;
				(* activ write *)
				ELSE
					(* copy profile to HDD data structure *)
					IF xFctCopyProfileToDataFile(	sNameOfProfile:=T_Profile.T_Id.sName,
													ptrStProzessData:=ADR(T_Profile.T_CopyProfileParameter.T_ProzessData),
													ptrOnlineChangeData:=ADR(T_Profile.T_CopyProfileParameter.T_ProfileOnlineChange),
													ptrDataFile:=ADR(T_HDD.T_Data)) 	THEN iStepFunction:=50; ELSE iStepFunction:=99; END_IF
					T_HDD.T_Ctrle.xLocked:=TRUE;
					(* next step *)
					xStepFunctionDone:=FALSE;
				END_IF
			ELSE
				(* activ error if time out done, HDD not ready *)
				IF TimerFileLocked.Q THEN
					 iStepFunction:=91;
				END_IF
			END_IF;
		(* waiting flag *)
		20:	IF T_HDD.T_Ctrle.xDone AND NOT(T_HDD.T_Ctrle.xErr) THEN iStepFunction:=30; END_IF
			IF T_HDD.T_Ctrle.xErr THEN iStepFunction:=80; END_IF
		(* copy value from HDD to Profile structure *)
		30:	FBCopyDataFileToProfile(	ptrStProzessData:=ADR(T_Profile.T_CopyProfileParameter.T_ProzessData),
									ptrOnlineChangeData:=ADR(T_Profile.T_CopyProfileParameter.T_ProfileOnlineChange),
									ptrDataFile:=ADR(T_HDD.T_Data),
									ptrNameOfProfile:=ADR(T_Profile.T_Ctrle.sProfileName));
			IF (FBCopyDataFileToProfile.bResultCopyData = 1) THEN
				iStepFunction:=90;
			ELSIF (FBCopyDataFileToProfile.bResultCopyData = 2) THEN
				iStepFunction:=98;
			END_IF
		(* activ write *)
		50:	sTmp:=CONCAT(sDriveName,T_Profile.T_Ctrle.sPathAndFileName);
			sTmp:=CONCAT(sTmp,'STATION');
			sTmp:=CONCAT(sTmp,UINT_TO_STRING(gciStationSt1));
			sTmp:=CONCAT(sTmp,'\');
			sTmp:=CONCAT(sTmp,INT_TO_STRING(T_Profile.T_Id.iNumber));
			sTmp:=CONCAT(sTmp,'.txt');
			T_HDD.T_File.sPathAndFileName:=sTmp;
			IF (T_Profile.T_Ctrle.iFunction = 2) THEN
				T_HDD.T_Ctrle.iFunction:=2;
			ELSE
				T_HDD.T_Ctrle.iFunction:=2;	(* 10 does not right function *)
			END_IF;
			T_HDD.T_Ctrle.xExecute:=TRUE;
			(* next step *)
			iStepFunction:=60;
			xStepFunctionDone:=FALSE;
		(* waiting flag *)
		60:	IF T_HDD.T_Ctrle.xDone AND NOT(T_HDD.T_Ctrle.xErr) THEN iStepFunction:=90; END_IF
			IF T_HDD.T_Ctrle.xErr THEN iStepFunction:=80; END_IF
		(* reset error *)
		80:	T_HDD.T_Ctrle.xReset:=TRUE;
			iStepFunction:=99;
		(* done *)
		90:	T_Profile.T_Ctrle.xDone:=TRUE;
			T_Profile.T_Ctrle.xErr:=FALSE;
			T_Profile.T_Ctrle.udiErrorID:=16#0;
			T_HDD.T_Ctrle.xExecute:=FALSE;
			T_HDD.T_Ctrle.xLocked:=FALSE;
			xReadProfile:=FALSE;
			xWriteProfile:=FALSE;
		(* start read error *)
		91:	T_Profile.T_Ctrle.xDone:=FALSE;
			T_Profile.T_Ctrle.xErr:=TRUE;
			T_Profile.T_Ctrle.udiErrorID:=16#F1000 + T_Profile.T_Ctrle.iFunction;
			T_HDD.T_Ctrle.xReset:=T_HDD.T_Ctrle.xErr;
			T_HDD.T_Ctrle.xExecute:=FALSE;
			T_HDD.T_Ctrle.xLocked:=FALSE;
			xReadProfile:=FALSE;
			xWriteProfile:=FALSE;
		(* syntax error *)
		98:	T_Profile.T_Ctrle.xDone:=FALSE;
			T_Profile.T_Ctrle.xErr:=TRUE;
			T_Profile.T_Ctrle.udiErrorID:=16#F2000;
			T_HDD.T_Ctrle.xReset:=T_HDD.T_Ctrle.xErr;
			T_HDD.T_Ctrle.xExecute:=FALSE;
			T_HDD.T_Ctrle.xLocked:=FALSE;
			xReadProfile:=FALSE;
			xWriteProfile:=FALSE;
		(* error *)
		99:	T_Profile.T_Ctrle.xDone:=FALSE;
			T_Profile.T_Ctrle.xErr:=TRUE;
			T_Profile.T_Ctrle.udiErrorID:=16#F1000 + T_Profile.T_Ctrle.iFunction;
			T_HDD.T_Ctrle.xReset:=T_HDD.T_Ctrle.xErr;
			T_HDD.T_Ctrle.xExecute:=FALSE;
			T_HDD.T_Ctrle.xLocked:=FALSE;
			xReadProfile:=FALSE;
			xWriteProfile:=FALSE;
		END_CASE
	END_IF

(* check if the USB stick exist *)
	IF xCheckUSBStick THEN
		CASE iStepFunction OF
		(* start timeout *)
		1:	TimerFileLocked(IN:=FALSE);
			iStepFunction:=2;
			sDriveName:='D:\';
		(* Überprüfe zuerst welchen Laufwerkbuchstabe das USB-Stick für Profile hat *)
		2:	IF T_HDD.T_Ctrle.xDone AND NOT(T_HDD.T_Ctrle.xErr) AND NOT(T_HDD.T_Ctrle.xLocked) THEN
				T_HDD.T_Ctrle.xLocked:=TRUE;
				(* next step *)
				iStepFunction:=iStepFunction + 1;
			ELSE
				(* activ error if time out done, HDD not ready *)
				IF TimerFileLocked.Q THEN
					 iStepFunction:=91;
				END_IF
			END_IF;
		(* Überprüfe zuerst welche USB Stick als CAQ definiert ist *)
		3:	IF NOT(gxHardwareOFF) THEN
				sTmp:='D:\PROFILE.txt';
			ELSE
				sTmp:='C:\PROFILE.txt';
			END_IF;
			T_HDD.T_File.sPathAndFileName:=sTmp;
			T_HDD.T_Ctrle.iFunction:=1;
			T_HDD.T_Ctrle.xExecute:=TRUE;
			(* next step *)
			iStepFunction:=iStepFunction + 1;
		(* waiting flag *)
		4:	IF T_HDD.T_Ctrle.xDone AND NOT(T_HDD.T_Ctrle.xErr) THEN
				iStepFunction:=10;
				IF NOT(gxHardwareOFF) THEN
					sDriveName:='D:\';
				ELSE
					sDriveName:='C:\';
				END_IF;
			END_IF
			IF T_HDD.T_Ctrle.xErr THEN T_HDD.T_Ctrle.xReset:=TRUE; iStepFunction:=iStepFunction + 1; END_IF
		5:	IF T_HDD.T_Ctrle.xDone AND NOT(T_HDD.T_Ctrle.xErr) THEN
				sTmp:='E:\PROFILE.txt';
				T_HDD.T_File.sPathAndFileName:=sTmp;
				T_HDD.T_Ctrle.iFunction:=1;
				T_HDD.T_Ctrle.xExecute:=TRUE;
				(* next step *)
				iStepFunction:=iStepFunction + 1;
			END_IF;
		(* waiting flag *)
		6:	IF T_HDD.T_Ctrle.xDone AND NOT(T_HDD.T_Ctrle.xErr) THEN iStepFunction:=10; sDriveName:='E:\'; END_IF
			IF T_HDD.T_Ctrle.xErr THEN T_HDD.T_Ctrle.xReset:=TRUE; iStepFunction:=99; END_IF
		(* start read *)
		10:	sTmp:=CONCAT(sDriveName,'PROFILETMP1234');
			(* create directory *)
			T_HDD.T_Ctrle.iFunction:=7;
			T_HDD.T_Ctrle.xLocked:=TRUE;
			T_HDD.T_File.sDirectoryPath:=sTmp;
			T_HDD.T_Ctrle.xExecute:=TRUE;
			(* next step *)
			iStepFunction:=20;
			xStepFunctionDone:=FALSE;
		(* waiting flag *)
		20:	IF T_HDD.T_Ctrle.xDone AND NOT(T_HDD.T_Ctrle.xErr) THEN iStepFunction:=30; END_IF
			IF T_HDD.T_Ctrle.xErr THEN T_HDD.T_Ctrle.xReset:=TRUE; iStepFunction:=30; END_IF
		(* waiting flag *)
		30:	IF T_HDD.T_Ctrle.xDone AND NOT(T_HDD.T_Ctrle.xErr) THEN
				sTmp:=CONCAT(sDriveName,'PROFILETMP1234');
				(* remove directory *)
				T_HDD.T_Ctrle.iFunction:=8;
				T_HDD.T_File.sDirectoryPath:=sTmp;
				T_HDD.T_Ctrle.xExecute:=TRUE;
				(* next step *)
				iStepFunction:=40;
				xStepFunctionDone:=FALSE;
			END_IF;
		(* waiting flag *)
		40:	IF T_HDD.T_Ctrle.xDone AND NOT(T_HDD.T_Ctrle.xErr) THEN iStepFunction:=90; END_IF
			IF T_HDD.T_Ctrle.xErr THEN T_HDD.T_Ctrle.xReset:=TRUE; iStepFunction:=99; END_IF
		(* done *)
		90:	T_Profile.T_Ctrle.xDone:=TRUE;
			T_Profile.T_Ctrle.xErr:=FALSE;
			T_Profile.T_Ctrle.udiErrorID:=16#0;
			T_HDD.T_Ctrle.xExecute:=FALSE;
			T_HDD.T_Ctrle.xLocked:=FALSE;
			xCheckUSBStick:=FALSE;
		(* start read error *)
		91:	T_Profile.T_Ctrle.xDone:=FALSE;
			T_Profile.T_Ctrle.xErr:=TRUE;
			T_Profile.T_Ctrle.udiErrorID:=16#F1000 + T_Profile.T_Ctrle.iFunction;
			T_HDD.T_Ctrle.xExecute:=FALSE;
			T_HDD.T_Ctrle.xLocked:=FALSE;
			xCheckUSBStick:=FALSE;
		(* start read error *)
		99:	T_Profile.T_Ctrle.xDone:=FALSE;
			T_Profile.T_Ctrle.xErr:=TRUE;
			T_Profile.T_Ctrle.udiErrorID:=16#FFFF;	(* USB-Stick does not exist *)
			T_HDD.T_Ctrle.xExecute:=FALSE;
			T_HDD.T_Ctrle.xLocked:=FALSE;
			xCheckUSBStick:=FALSE;
		END_CASE;
	END_IF;

(* Read liste profile station *)
	IF xReadProfileListeStation THEN
		CASE iStepFunction OF
		(* start timeout *)
		1:	TimerFileLocked(IN:=FALSE);
			iStepFunction:=10;
		(* start read *)
		10:	IF T_HDD.T_Ctrle.xDone AND NOT(T_HDD.T_Ctrle.xErr) AND NOT(T_HDD.T_Ctrle.xLocked) THEN
				(* Init. value *)
				iProfileNr:=1;
				T_Profile.T_IDProfileStation:=T_DeleteIDProfileStation;
				FOR jj:=1 TO csiMaxProfile DO
					T_Profile.T_IDProfileStation[jj].iNumber:=jj;
					T_Profile.T_IDProfileStation[jj].sName:='';
				END_FOR;
				T_Profile.T_IDProfileStation[1].iNumber:=1;
				T_Profile.T_IDProfileStation[1].sName:='Default';
				(* next step *)
				iStepFunction:=20;
				xStepFunctionDone:=FALSE;
				T_HDD.T_Ctrle.xLocked:=TRUE;
			ELSE
				(* activ error if time out done, HDD not ready *)
				IF TimerFileLocked.Q THEN
					 iStepFunction:=91;
				END_IF
			END_IF;
		20:	T_HDD.T_Data.sData:=sDeleteData;
			sTmp:=CONCAT(sDriveName,T_Profile.T_Ctrle.sPathAndFileName);
			sTmp:=CONCAT(sTmp,'STATION');
			sTmp:=CONCAT(sTmp,UINT_TO_STRING(gciStationSt1));
			sTmp:=CONCAT(sTmp,'\');
			sTmp:=CONCAT(sTmp,INT_TO_STRING(iProfileNr));
			sTmp:=CONCAT(sTmp,'.txt');
			(* read file only 1 line *)
			T_HDD.T_Ctrle.iFunction:=11;
			T_HDD.T_File.sPathAndFileName:=sTmp;
			T_HDD.T_Ctrle.xExecute:=TRUE;
			(* next step *)
			iStepFunction:=30;
			xStepFunctionDone:=FALSE;
		(* waiting flag *)
		30:	IF T_HDD.T_Ctrle.xDone AND NOT(T_HDD.T_Ctrle.xErr) THEN
				T_Profile.T_IDProfileStation[iProfileNr].iNumber:=iProfileNr;
				sTmp:=T_HDD.T_Data.sData[1];
				sTmp:=sFctDeleteChar(sString:=sTmp, sChar:='$N');
				sTmp:=sFctDeleteChar(sString:=sTmp, sChar:='$L');
				sTmp:=sFctDeleteChar(sString:=sTmp, sChar:=' ');
				IF (FIND(sTmp,';') > 0) THEN
					iFindChar:=FIND(sTmp,';');
					sTmp:=MID(STR:=sTmp,LEN:=iFindChar - 1,POS:=1);
				END_IF;
				T_Profile.T_IDProfileStation[iProfileNr].sName:=sTmp;
				iStepFunction:=35;
			END_IF
			IF T_HDD.T_Ctrle.xErr THEN
				T_HDD.T_Ctrle.xReset:=T_HDD.T_Ctrle.xErr;
				T_Profile.T_IDProfileStation[iProfileNr].iNumber:=iProfileNr;
				T_Profile.T_IDProfileStation[iProfileNr].sName:='';
				iStepFunction:=35;
			END_IF
		(* next file *)
		35:	IF iProfileNr < csiMaxProfile THEN
				iProfileNr:=iProfileNr+1; iStepFunction:=20;
			ELSE
				iStepFunction:=90;
			END_IF
		(* reset HDD error *)
		80:	T_HDD.T_Ctrle.xReset:=T_HDD.T_Ctrle.xErr;
			iStepFunction:=99;
		(* done *)
		90:	T_Profile.T_Ctrle.xDone:=TRUE;
			T_Profile.T_Ctrle.xErr:=FALSE;
			T_Profile.T_Ctrle.udiErrorID:=16#0;
			T_HDD.T_Ctrle.xExecute:=FALSE;
			T_HDD.T_Ctrle.xLocked:=FALSE;
			xReadProfileListeStation:=FALSE;
		(* start read error *)
		91:	T_Profile.T_Ctrle.xDone:=FALSE;
			T_Profile.T_Ctrle.xErr:=TRUE;
			T_Profile.T_Ctrle.udiErrorID:=16#F1000 + T_Profile.T_Ctrle.iFunction;
			T_HDD.T_Ctrle.xExecute:=FALSE;
			T_HDD.T_Ctrle.xLocked:=FALSE;
			xReadProfileListeStation:=FALSE;
		(* error *)
		99:	T_Profile.T_Ctrle.xDone:=FALSE;
			T_Profile.T_Ctrle.xErr:=TRUE;
			T_Profile.T_Ctrle.udiErrorID:=16#F1000 + T_Profile.T_Ctrle.iFunction;
			T_HDD.T_Ctrle.xExecute:=FALSE;
			T_HDD.T_Ctrle.xLocked:=FALSE;
			xReadProfileListeStation:=FALSE;
		END_CASE
	END_IF

	IF xCreateDefaultProfile THEN
		CASE iStepFunction OF
		(* start timeout *)
		1:	TimerFileLocked(IN:=FALSE);
			iStepFunction:=10;
		(* start read *)
		10:	IF T_HDD.T_Ctrle.xDone AND NOT(T_HDD.T_Ctrle.xErr) AND NOT(T_HDD.T_Ctrle.xLocked) THEN
				(* next step *)
				iStepFunction:=20;
				xStepFunctionDone:=FALSE;
				T_HDD.T_Ctrle.xLocked:=TRUE;
			ELSE
				(* activ error if time out done, HDD not ready *)
				IF TimerFileLocked.Q THEN
					 iStepFunction:=91;
				END_IF
			END_IF;
		20:	T_HDD.T_Data.sData:=sDeleteData;
			xFctSetDefaultValueStaticProfile(	ptrT_DefaultProfileParameter:=ADR(T_Profile.T_DefaultProfileParameter));
			xFctCopyProfileToDataFile(	sNameOfProfile:='Default',
									ptrStProzessData:=ADR(T_Profile.T_DefaultProfileParameter.T_ProzessData),
									ptrOnlineChangeData:=ADR(T_Profile.T_DefaultProfileParameter.T_ProfileOnlineChange),
									ptrDataFile:=ADR(T_HDD.T_Data));
			sTmp:=CONCAT(sDriveName,T_Profile.T_Ctrle.sPathAndFileName);
			sTmp:=CONCAT(sTmp,'1');
			sTmp:=CONCAT(sTmp,'.txt');
			(* write file complete *)
			T_HDD.T_Ctrle.iFunction:=2;	(* 10 does not right function *)
			T_HDD.T_File.sPathAndFileName:=sTmp;
			T_HDD.T_Ctrle.xExecute:=TRUE;
			(* next step *)
			iStepFunction:=30;
			xStepFunctionDone:=FALSE;
		(* waiting flag *)
		30:	IF T_HDD.T_Ctrle.xDone AND NOT(T_HDD.T_Ctrle.xErr) THEN
				T_Profile.T_IDProfileStation[1].iNumber:=1;
				T_Profile.T_IDProfileStation[1].sName:='Default';
				iStepFunction:=90;
			END_IF
			IF T_HDD.T_Ctrle.xErr THEN
				T_HDD.T_Ctrle.xReset:=T_HDD.T_Ctrle.xErr;
				iStepFunction:=35;
			END_IF
		(* try to create first level directory *)
		35:	IF T_HDD.T_Ctrle.xDone THEN
				sTmp:=CONCAT(sDriveName,T_Profile.T_Ctrle.sPathAndFileName);
				(* create directory *)
				T_HDD.T_Ctrle.iFunction:=7;
				T_HDD.T_Ctrle.xLocked:=TRUE;
				T_HDD.T_File.sDirectoryPath:=sTmp;
				T_HDD.T_Ctrle.xExecute:=TRUE;
				(* next step *)
				iStepFunction:=36;
				xStepFunctionDone:=FALSE;
			END_IF;
		(* waiting flag *)
		36:	IF T_HDD.T_Ctrle.xDone AND NOT(T_HDD.T_Ctrle.xErr) THEN
				iStepFunction:=37;
			END_IF
			IF T_HDD.T_Ctrle.xErr THEN
				T_HDD.T_Ctrle.xReset:=T_HDD.T_Ctrle.xErr;
				iStepFunction:=37;
			END_IF
		(* try to create second level directory *)
		37:	IF T_HDD.T_Ctrle.xDone THEN
				sTmp:=T_Profile.T_Ctrle.sPathAndFileName;
				sTmp:=CONCAT(sTmp,'PROFILE');
				(* create directory *)
				T_HDD.T_Ctrle.iFunction:=7;
				T_HDD.T_Ctrle.xLocked:=TRUE;
				T_HDD.T_File.sDirectoryPath:=sTmp;
				T_HDD.T_Ctrle.xExecute:=TRUE;
				(* next step *)
				iStepFunction:=38;
				xStepFunctionDone:=FALSE;
			END_IF;
		(* waiting flag *)
		38:	IF T_HDD.T_Ctrle.xDone AND NOT(T_HDD.T_Ctrle.xErr) THEN
				iStepFunction:=20;
			END_IF
			IF T_HDD.T_Ctrle.xErr THEN
				T_HDD.T_Ctrle.xReset:=T_HDD.T_Ctrle.xErr;
				iStepFunction:=99;
			END_IF
		(* reset HDD error *)
		80:	T_HDD.T_Ctrle.xReset:=T_HDD.T_Ctrle.xErr;
			iStepFunction:=99;
		(* done *)
		90:	T_Profile.T_Ctrle.xDone:=TRUE;
			T_Profile.T_Ctrle.xErr:=FALSE;
			T_Profile.T_Ctrle.udiErrorID:=16#0;
			T_HDD.T_Ctrle.xExecute:=FALSE;
			T_HDD.T_Ctrle.xLocked:=FALSE;
			xCreateDefaultProfile:=FALSE;
		(* start read error *)
		91:	T_Profile.T_Ctrle.xDone:=FALSE;
			T_Profile.T_Ctrle.xErr:=TRUE;
			T_Profile.T_Ctrle.udiErrorID:=16#F1000 + T_Profile.T_Ctrle.iFunction;
			T_HDD.T_Ctrle.xExecute:=FALSE;
			T_HDD.T_Ctrle.xLocked:=FALSE;
			xCreateDefaultProfile:=FALSE;
		(* error *)
		99:	T_Profile.T_Ctrle.xDone:=FALSE;
			T_Profile.T_Ctrle.xErr:=TRUE;
			T_Profile.T_Ctrle.udiErrorID:=16#F1000 + T_Profile.T_Ctrle.iFunction;
			T_HDD.T_Ctrle.xExecute:=FALSE;
			T_HDD.T_Ctrle.xLocked:=FALSE;
			xCreateDefaultProfile:=FALSE;
		END_CASE
	END_IF;

(* Delete profile *)
	IF xDeleteProfile THEN
		CASE iStepFunction OF
		(* check if HDD state *)
		(* start timeout *)
		1:	TimerFileLocked(IN:=FALSE);
			iStepFunction:=10;
		(* file name and activ read or write *)
		10:	IF T_HDD.T_Ctrle.xDone AND NOT(T_HDD.T_Ctrle.xErr) AND NOT(T_HDD.T_Ctrle.xLocked) THEN
				sTmp:=CONCAT(sDriveName,T_Profile.T_Ctrle.sPathAndFileName);
				sTmp:=CONCAT(sTmp,'STATION');
				sTmp:=CONCAT(sTmp,UINT_TO_STRING(gciStationSt1));
				sTmp:=CONCAT(sTmp,'\');
				sTmp:=CONCAT(sTmp,INT_TO_STRING(T_Profile.T_Id.iNumber));
				sTmp:=CONCAT(sTmp,'.txt');
				T_HDD.T_Ctrle.iFunction:=5;	(* Delete Profile *)
				T_HDD.T_Ctrle.xLocked:=TRUE;
				T_HDD.T_File.sPathAndFileName:=sTmp;
				T_HDD.T_Ctrle.xExecute:=TRUE;
				T_Profile.T_Ctrle.sProfileName:='';
				(* next step *)
				iStepFunction:=20;
				xStepFunctionDone:=FALSE;
			ELSE
				(* activ error if time out done, HDD not ready *)
				IF TimerFileLocked.Q THEN
					 iStepFunction:=91;
				END_IF
			END_IF;
		(* waiting flag *)
		20:	IF NOT(T_HDD.T_Ctrle.xExecute) AND T_HDD.T_Ctrle.xDone AND NOT(T_HDD.T_Ctrle.xErr) THEN iStepFunction:=90; END_IF
			IF NOT(T_HDD.T_Ctrle.xExecute) AND T_HDD.T_Ctrle.xErr THEN iStepFunction:=80; END_IF
		(* reset error *)
		80:	T_HDD.T_Ctrle.xReset:=TRUE;
			iStepFunction:=99;
		(* done *)
		90:	T_Profile.T_Ctrle.xDone:=TRUE;
			T_Profile.T_Ctrle.xErr:=FALSE;
			T_Profile.T_Ctrle.udiErrorID:=16#0;
			T_HDD.T_Ctrle.xExecute:=FALSE;
			T_HDD.T_Ctrle.xLocked:=FALSE;
			xDeleteProfile:=FALSE;
		(* start read error *)
		91:	T_Profile.T_Ctrle.xDone:=FALSE;
			T_Profile.T_Ctrle.xErr:=TRUE;
			T_Profile.T_Ctrle.udiErrorID:=16#F1000 + T_Profile.T_Ctrle.iFunction;
			T_HDD.T_Ctrle.xReset:=T_HDD.T_Ctrle.xErr;
			T_HDD.T_Ctrle.xExecute:=FALSE;
			T_HDD.T_Ctrle.xLocked:=FALSE;
			xDeleteProfile:=FALSE;
		(* error *)
		99:	T_Profile.T_Ctrle.xDone:=FALSE;
			T_Profile.T_Ctrle.xErr:=TRUE;
			T_Profile.T_Ctrle.udiErrorID:=16#F1000 + T_Profile.T_Ctrle.iFunction;
			T_HDD.T_Ctrle.xReset:=T_HDD.T_Ctrle.xErr;
			T_HDD.T_Ctrle.xExecute:=FALSE;
			T_HDD.T_Ctrle.xLocked:=FALSE;
			xDeleteProfile:=FALSE;
		END_CASE
	END_IF

	IF xRenameProfile THEN
		CASE iStepFunction OF
		(* start timeout *)
		1:	TimerFileLocked(IN:=FALSE);
			iStepFunction:=10;
		(* start read *)
		10:	IF T_HDD.T_Ctrle.xDone AND NOT(T_HDD.T_Ctrle.xErr) AND NOT(T_HDD.T_Ctrle.xLocked) THEN
				T_HDD.T_Data.sData:=sDeleteData;
				sTmp:=CONCAT(sDriveName,T_Profile.T_Ctrle.sPathAndFileName);
				sTmp:=CONCAT(sTmp,'STATION');
				sTmp:=CONCAT(sTmp,UINT_TO_STRING(gciStationSt1));
				sTmp:=CONCAT(sTmp,'\');
				sTmp:=CONCAT(sTmp,INT_TO_STRING(T_Profile.T_Id.iNumber));
				sTmp:=CONCAT(sTmp,'.txt');
				T_HDD.T_Ctrle.iFunction:=1;	(* Read Profile, 9 does not right function *)
				T_HDD.T_Ctrle.xLocked:=TRUE;
				T_HDD.T_File.sPathAndFileName:=sTmp;
				T_HDD.T_Ctrle.xExecute:=TRUE;
				T_Profile.T_Ctrle.sProfileName:='';
				(* next step *)
				iStepFunction:=20;
				xStepFunctionDone:=FALSE;
			ELSE
				(* activ error if time out done, HDD not ready *)
				IF TimerFileLocked.Q THEN
					 iStepFunction:=91;
				END_IF
			END_IF;
		(* waiting flag *)
		20:	IF NOT(T_HDD.T_Ctrle.xExecute) AND T_HDD.T_Ctrle.xDone AND NOT(T_HDD.T_Ctrle.xErr) THEN
				FBCopyDataFileToProfile(	ptrStProzessData:=ADR(T_Profile.T_LoadProfileParameter.T_ProzessData),
										ptrOnlineChangeData:=ADR(T_Profile.T_LoadProfileParameter.T_ProfileOnlineChange),
										ptrDataFile:=ADR(T_HDD.T_Data),
										ptrNameOfProfile:=ADR(T_Profile.T_Ctrle.sProfileName));
				IF (FBCopyDataFileToProfile.bResultCopyData = 1) THEN
					iStepFunction:=30;
				ELSIF (FBCopyDataFileToProfile.bResultCopyData = 2) THEN
					iStepFunction:=98;
				END_IF
			END_IF
			IF NOT(T_HDD.T_Ctrle.xExecute) AND T_HDD.T_Ctrle.xErr THEN
				iStepFunction:=80;
			END_IF
		30:	(* copy profile to HDD data structure *)
			IF xFctCopyProfileToDataFile(	sNameOfProfile:=T_Profile.T_Id.sName,
										ptrStProzessData:=ADR(T_Profile.T_LoadProfileParameter.T_ProzessData),
										ptrOnlineChangeData:=ADR(T_Profile.T_LoadProfileParameter.T_ProfileOnlineChange),
										ptrDataFile:=ADR(T_HDD.T_Data)) 	THEN iStepFunction:=40; ELSE iStepFunction:=99; END_IF
			sTmp:=CONCAT(sDriveName,T_Profile.T_Ctrle.sPathAndFileName);
			sTmp:=CONCAT(sTmp,'STATION');
			sTmp:=CONCAT(sTmp,UINT_TO_STRING(gciStationSt1));
			sTmp:=CONCAT(sTmp,'\');
			sTmp:=CONCAT(sTmp,INT_TO_STRING(T_Profile.T_Id.iNumber));
			sTmp:=CONCAT(sTmp,'.txt');
			(* write file  *)
			T_HDD.T_Ctrle.iFunction:=2;	(* 10 does not right function *)
			T_HDD.T_File.sPathAndFileName:=sTmp;
			T_HDD.T_Ctrle.xExecute:=TRUE;
			(* next step *)
			iStepFunction:=40;
			xStepFunctionDone:=FALSE;
		(* waiting flag *)
		40:	IF NOT(T_HDD.T_Ctrle.xExecute) AND T_HDD.T_Ctrle.xDone AND NOT(T_HDD.T_Ctrle.xErr) THEN
				iStepFunction:=90;
			END_IF
			IF NOT(T_HDD.T_Ctrle.xExecute) AND T_HDD.T_Ctrle.xErr THEN
				iStepFunction:=80;
			END_IF
		(* reset HDD error *)
		80:	T_HDD.T_Ctrle.xReset:=T_HDD.T_Ctrle.xErr;
			iStepFunction:=99;
		(* done *)
		90:	T_Profile.T_Ctrle.xDone:=TRUE;
			T_Profile.T_Ctrle.xErr:=FALSE;
			T_Profile.T_Ctrle.udiErrorID:=16#0;
			T_HDD.T_Ctrle.xExecute:=FALSE;
			T_HDD.T_Ctrle.xLocked:=FALSE;
			xRenameProfile:=FALSE;
		(* start read error *)
		91:	T_Profile.T_Ctrle.xDone:=FALSE;
			T_Profile.T_Ctrle.xErr:=TRUE;
			T_Profile.T_Ctrle.udiErrorID:=16#F1000 + T_Profile.T_Ctrle.iFunction;
			T_HDD.T_Ctrle.xExecute:=FALSE;
			T_HDD.T_Ctrle.xLocked:=FALSE;
			xRenameProfile:=FALSE;
		(* syntax error *)
		98:	T_Profile.T_Ctrle.xDone:=FALSE;
			T_Profile.T_Ctrle.xErr:=TRUE;
			T_Profile.T_Ctrle.udiErrorID:=16#F2000;
			T_HDD.T_Ctrle.xReset:=T_HDD.T_Ctrle.xErr;
			T_HDD.T_Ctrle.xExecute:=FALSE;
			T_HDD.T_Ctrle.xLocked:=FALSE;
			xRenameProfile:=FALSE;
		(* error *)
		99:	T_Profile.T_Ctrle.xDone:=FALSE;
			T_Profile.T_Ctrle.xErr:=TRUE;
			T_Profile.T_Ctrle.udiErrorID:=16#F1000 + T_Profile.T_Ctrle.iFunction;
			T_HDD.T_Ctrle.xExecute:=FALSE;
			T_HDD.T_Ctrle.xLocked:=FALSE;
			xRenameProfile:=FALSE;
		END_CASE
	END_IF;
END_FUNCTION_BLOCK

(* POU GENERAL/PROFILE/FB_CopyDataFileToProfile, ST *)
FUNCTION_BLOCK FB_CopyDataFileToProfile
VAR_INPUT
	ptrStProzessData:POINTER TO ST_EXCHG_PARAM_STANDARDPROCESS;
	ptrOnlineChangeData:POINTER TO ST_PROFILEONLINECHANGE_DATA;
	ptrDataFile:POINTER TO ARRAY[1..csiMaxFileLine] OF STRING(csiMaxCharPerLine);
	ptrNameOfProfile:POINTER TO STRING(30);
END_VAR
VAR_OUTPUT
	bResultCopyData:BYTE;
END_VAR
VAR
(* variable *)
	i:INT;
	iPosStartCarValue:INT;
	iPosStopCarValue:INT;
	sValue:STRING;
	sVariableName:STRING;
(* Tmp variable *)
	sTmp:STRING;
	iCountParameter: INT;
	xWrongSyntax: BOOL;
	iFindChar: INT;
	iStepCopy: INT;
END_VAR
(* Wegen Zykluszeitüberschreitung wurde nun neu ein FB erstellt und das Überprüfen unterteilt *)
CASE iStepCopy OF
0:	(* Init. variable *)
	bResultCopyData:=0;
	xWrongSyntax:=FALSE;
	sTmp:=ptrDataFile^[1];
	sTmp:=sFctDeleteChar(sString:=sTmp, sChar:='$N');
	sTmp:=sFctDeleteChar(sString:=sTmp, sChar:='$L');
	sTmp:=sFctDeleteChar(sString:=sTmp, sChar:=' ');
	IF (FIND(sTmp,';') > 0) THEN
		iFindChar:=FIND(sTmp,';');
		sTmp:=MID(STR:=sTmp,LEN:=iFindChar - 1,POS:=1);
	END_IF;
	ptrNameOfProfile^:=sTmp;
	iCountParameter:=0;
	iStepCopy:=iStepCopy + 1;
1:	FOR i:= 1 TO ciMaxProfileParameter DO
		CheckParameter;
	END_FOR
	iStepCopy:=99;
99:	IF (iCountParameter <> csiMaxProfileParameter) THEN
		xWrongSyntax:=TRUE;
	END_IF;
	(* confirm copy value *)
	IF NOT(xWrongSyntax) THEN
		bResultCopyData:=1;
	ELSE
		bResultCopyData:=2;
	END_IF;
	iStepCopy:=0;
END_CASE;
END_FUNCTION_BLOCK
ACTION CheckParameter:
sTmp:=ptrDataFile^[i];
sTmp:=sFctDeleteChar(sString:=sTmp, sChar:='$N');
sTmp:=sFctDeleteChar(sString:=sTmp, sChar:='$L');
sTmp:=sFctDeleteChar(sString:=sTmp, sChar:=' ');
IF FIND(sTmp,':=') <> 0 THEN
(* read value *)
	iPosStartCarValue:= FIND(sTmp,':=')+2;
	iPosStopCarValue:= FIND(sTmp,';');
	sValue:=MID(sTmp,iPosStopCarValue - iPosStartCarValue,iPosStartCarValue);

	IF (sFctUpLowCase(xLowConvert:=TRUE, sInString:=sValue) <> 'false') AND (sFctUpLowCase(xLowConvert:=TRUE, sInString:=sValue) <> 'true') THEN
		IF NOT(xFctCheckNumber(sValue:=sValue,xAlowDoubleSign:=FALSE)) THEN
			xWrongSyntax:=TRUE;
		END_IF;
	END_IF;
(* read variable name *)
	IF NOT(xWrongSyntax) THEN
		iPosStartCarValue:= FIND(sTmp,':')+1;
		iPosStopCarValue:= FIND(sTmp,':=');
		sVariableName:=sFctUpLowCase(	xLowConvert:=TRUE,
										sInString:=MID(sTmp,iPosStopCarValue - iPosStartCarValue,iPosStartCarValue));

		IF sVariableName = 'rtorquelevelhc' THEN ptrOnlineChangeData^.rTorqueLevelHC:=STRING_TO_REAL(sValue); iCountParameter:=iCountParameter + 1;
		ELSIF sVariableName = 'rforcedeflection' THEN ptrOnlineChangeData^.rForceDeflection:=STRING_TO_REAL(sValue); iCountParameter:=iCountParameter + 1;
		ELSIF sVariableName = 'rworkingspeedforward' THEN ptrOnlineChangeData^.rWorkingSpeedForward:=STRING_TO_REAL(sValue); iCountParameter:=iCountParameter + 1;
		ELSIF sVariableName = 'rworkingoffsetbackward' THEN ptrOnlineChangeData^.rWorkingOffsetBackward:=STRING_TO_REAL(sValue); iCountParameter:=iCountParameter + 1;
		ELSIF sVariableName = 'rworkingspeedbackward' THEN ptrOnlineChangeData^.rWorkingSpeedBackward:=STRING_TO_REAL(sValue); iCountParameter:=iCountParameter + 1;
		ELSIF sVariableName = 'rworkingspindlespeed' THEN ptrOnlineChangeData^.rWorkingSpindleSpeed:=STRING_TO_REAL(sValue); iCountParameter:=iCountParameter + 1;

		ELSIF sVariableName = 'rpositionload' THEN ptrStProzessData^.rPositionLoad:=STRING_TO_REAL(sValue); iCountParameter:=iCountParameter + 1;
		ELSIF sVariableName = 'rpositionstartproc' THEN ptrStProzessData^.rPositionStartProc:=STRING_TO_REAL(sValue); iCountParameter:=iCountParameter + 1;
		ELSIF sVariableName = 'rpositionendproc' THEN ptrStProzessData^.rPositionEndProc:=STRING_TO_REAL(sValue); iCountParameter:=iCountParameter + 1;
		ELSIF sVariableName = 'rpositiontoolchange' THEN ptrStProzessData^.rPositionToolChange:=STRING_TO_REAL(sValue); iCountParameter:=iCountParameter + 1;
		ELSIF sVariableName = 'rinfeedzaxisspeed' THEN ptrStProzessData^.rInfeedZAxisSpeed:=STRING_TO_REAL(sValue); iCountParameter:=iCountParameter + 1;
		ELSIF sVariableName = 'rinfeedspindlespeed' THEN ptrStProzessData^.rInfeedSpindleSpeed:=STRING_TO_REAL(sValue); iCountParameter:=iCountParameter + 1;
		ELSIF sVariableName = 'routfeedstrokeaxisspeed' THEN ptrStProzessData^.rOutfeedStrokeAxisSpeed:=STRING_TO_REAL(sValue); iCountParameter:=iCountParameter + 1;
		ELSIF sVariableName = 'routfeedspindlespeed' THEN ptrStProzessData^.rOutfeedSpindleSpeed:=STRING_TO_REAL(sValue); iCountParameter:=iCountParameter + 1;
		ELSIF sVariableName = 'rinfeedforcedeflection' THEN ptrStProzessData^.rInfeedForceDeflection:=STRING_TO_REAL(sValue); iCountParameter:=iCountParameter + 1;
		ELSIF sVariableName = 'rinfeedoffsetbackward' THEN ptrStProzessData^.rInfeedOffsetBackward:=STRING_TO_REAL(sValue); iCountParameter:=iCountParameter + 1;
		ELSIF sVariableName = 'inumbertryinfeed' THEN ptrStProzessData^.iNumberTryInfeed:=STRING_TO_INT(sValue); iCountParameter:=iCountParameter + 1;

		ELSIF sVariableName = 'rprocessmintime' THEN ptrStProzessData^.rProcessMinTime:=STRING_TO_REAL(sValue); iCountParameter:=iCountParameter + 1;
		ELSIF sVariableName = 'rprocessmaxtime' THEN ptrStProzessData^.rProcessMaxTime:=STRING_TO_REAL(sValue); iCountParameter:=iCountParameter + 1;
		ELSIF sVariableName = 'ihcstartprocposcounter' THEN ptrStProzessData^.iHCStartProcPosCounter:=STRING_TO_INT(sValue); iCountParameter:=iCountParameter + 1;
		ELSIF sVariableName = 'rdeflectionsensoroffset' THEN ptrStProzessData^.rDeflectionSensorOffset:=STRING_TO_REAL(sValue); iCountParameter:=iCountParameter + 1;
		ELSIF sVariableName = 'rtorquelevel_overload' THEN ptrStProzessData^.rTorqueLevel_Overload:=STRING_TO_REAL(sValue); iCountParameter:=iCountParameter + 1;

		ELSIF sVariableName = 'isparkoutstrokecount' THEN ptrStProzessData^.iSparkOutStrokeCount:=STRING_TO_INT(sValue); iCountParameter:=iCountParameter + 1;
		ELSIF sVariableName = 'rsparkoutstrokelength' THEN ptrStProzessData^.rSparkOutStrokeLength:=STRING_TO_REAL(sValue); iCountParameter:=iCountParameter + 1;
		ELSIF sVariableName = 'rsparkoutstrokespeed' THEN ptrStProzessData^.rSparkOutStrokeSpeed:=STRING_TO_REAL(sValue); iCountParameter:=iCountParameter + 1;
		ELSIF sVariableName = 'rsparkoutforcedeflection' THEN ptrStProzessData^.rSparkOutForceDeflection:=STRING_TO_REAL(sValue); iCountParameter:=iCountParameter + 1;
		ELSIF sVariableName = 'rsparkouttorquelevel' THEN ptrStProzessData^.rSparkOutTorqueLevel:=STRING_TO_REAL(sValue); iCountParameter:=iCountParameter + 1;

		ELSIF sVariableName = 'rpostoolguid_up' THEN ptrStProzessData^.rPosToolGuid_Up:=STRING_TO_REAL(sValue); iCountParameter:=iCountParameter + 1;
		ELSIF sVariableName = 'rpostoolguid_down' THEN ptrStProzessData^.rPosToolGuid_Down:=STRING_TO_REAL(sValue); iCountParameter:=iCountParameter + 1;
		ELSIF sVariableName = 'rdistancetoolguide' THEN ptrStProzessData^.rDistanceToolGuide:=STRING_TO_REAL(sValue); iCountParameter:=iCountParameter + 1;
		ELSIF sVariableName = 'rdistancetoolendpos' THEN ptrStProzessData^.rDistanceToolEndPos:=STRING_TO_REAL(sValue); iCountParameter:=iCountParameter + 1;
		ELSIF sVariableName = 'rlengthtool_fixed' THEN ptrStProzessData^.rLengthTool_Fixed:=STRING_TO_REAL(sValue); iCountParameter:=iCountParameter + 1;
		ELSIF sVariableName = 'rlengthtool_work' THEN ptrStProzessData^.rLengthTool_Work:=STRING_TO_REAL(sValue); iCountParameter:=iCountParameter + 1;
		ELSIF sVariableName = 'rlengthtoolguide' THEN ptrStProzessData^.rLengthToolGuide:=STRING_TO_REAL(sValue); iCountParameter:=iCountParameter + 1;
		ELSIF sVariableName = 'rlengthairtableboard' THEN ptrStProzessData^.rLengthAirTableBoard:=STRING_TO_REAL(sValue); iCountParameter:=iCountParameter + 1;
		ELSIF sVariableName = 'xconfigactive' THEN ptrStProzessData^.xConfigActive:=STRING_TO_BOOL(sValue); iCountParameter:=iCountParameter + 1;

		ELSIF sVariableName = 'imaxtorque' THEN ptrStProzessData^.iMaxTorque:=STRING_TO_INT(sValue); iCountParameter:=iCountParameter + 1;
		ELSIF sVariableName = 'rspeedzaxisforbackward' THEN ptrStProzessData^.rSpeedZAxisForBackward:=STRING_TO_REAL(sValue); iCountParameter:=iCountParameter + 1;
		ELSIF sVariableName = 'rworkingspeedoscillation' THEN ptrStProzessData^.rWorkingSpeedOscillation:=STRING_TO_INT(sValue); iCountParameter:=iCountParameter + 1;
		ELSIF sVariableName = 'rz1axisposswitchoaxisoff' THEN ptrStProzessData^.rZ1AxisPosSwitchOAxisOff:=STRING_TO_INT(sValue); iCountParameter:=iCountParameter + 1;
		ELSIF sVariableName = 'xactivatecoolantprocess' THEN ptrStProzessData^.xActivateCoolantProcess:=STRING_TO_BOOL(sValue); iCountParameter:=iCountParameter + 1;
		ELSIF sVariableName = 'rstrokeaxisposswitchcoolantoff' THEN ptrStProzessData^.rStrokeAxisPosSwitchCoolantOff:=STRING_TO_INT(sValue); iCountParameter:=iCountParameter + 1;

		ELSIF sVariableName = 'rcentringposz1axis' THEN ptrStProzessData^.rCentringPosZ1Axis:=STRING_TO_REAL(sValue); iCountParameter:=iCountParameter + 1;
		ELSIF sVariableName = 'rcentringposspeedslowz1axis' THEN ptrStProzessData^.rCentringPosSpeedSlowZ1Axis:=STRING_TO_REAL(sValue); iCountParameter:=iCountParameter + 1;
		ELSIF sVariableName = 'rcentringposspeedfastz1axis' THEN ptrStProzessData^.rCentringPosSpeedFastZ1Axis:=STRING_TO_REAL(sValue); iCountParameter:=iCountParameter + 1;
		ELSIF sVariableName = 'rcentringspeedsaxis' THEN ptrStProzessData^.rCentringSpeedSAxis:=STRING_TO_REAL(sValue); iCountParameter:=iCountParameter + 1;
		ELSIF sVariableName = 'rcentringspeedoaxis' THEN ptrStProzessData^.rCentringSpeedOAxis:=STRING_TO_REAL(sValue); iCountParameter:=iCountParameter + 1;
		ELSIF sVariableName = 'rcentringbackstrokeoffsetfirsthc' THEN ptrStProzessData^.rCentringBackStrokeOffsetFirstHC:=STRING_TO_REAL(sValue); iCountParameter:=iCountParameter + 1;
		ELSIF sVariableName = 'rcentringbackstrokeoffsetafterfirsthc' THEN ptrStProzessData^.rCentringBackStrokeOffsetAfterFirstHC:=STRING_TO_REAL(sValue); iCountParameter:=iCountParameter + 1;
		ELSIF sVariableName = 'rcentringoffsetbeforelasthc' THEN ptrStProzessData^.rCentringOffsetBeforeLastHC:=STRING_TO_REAL(sValue); iCountParameter:=iCountParameter + 1;
		ELSIF sVariableName = 'rcentringbackstrokespeed' THEN ptrStProzessData^.rCentringBackStrokeSpeed:=STRING_TO_REAL(sValue); iCountParameter:=iCountParameter + 1;
		ELSIF sVariableName = 'rcentringtimehcactive' THEN ptrStProzessData^.rCentringTimeHCActive:=STRING_TO_REAL(sValue); iCountParameter:=iCountParameter + 1;
		ELSIF sVariableName = 'rcentringtimehcinactive' THEN ptrStProzessData^.rCentringTimeHCInactive:=STRING_TO_REAL(sValue); iCountParameter:=iCountParameter + 1;
		ELSIF sVariableName = 'icentringnumbermaxhcinwindow' THEN ptrStProzessData^.iCentringNumberMaxHCinWindow:=STRING_TO_INT(sValue); iCountParameter:=iCountParameter + 1;
		ELSIF sVariableName = 'rcentringhcwindow' THEN ptrStProzessData^.rCentringHCWindow:=STRING_TO_REAL(sValue); iCountParameter:=iCountParameter + 1;
		ELSIF sVariableName = 'rcentringforcedeflection' THEN ptrStProzessData^.rCentringForceDeflection:=STRING_TO_REAL(sValue); iCountParameter:=iCountParameter + 1;
		ELSIF sVariableName = 'rcentringoffsetbackward' THEN ptrStProzessData^.rCentringOffsetBackward:=STRING_TO_REAL(sValue); iCountParameter:=iCountParameter + 1;
		ELSIF sVariableName = 'rcenteringdeflectionsensoroffset' THEN ptrStProzessData^.rCenteringDeflectionSensorOffset:=STRING_TO_REAL(sValue); iCountParameter:=iCountParameter + 1;
		ELSIF sVariableName = 'rcentringoffsetslowtofastzspeed' THEN ptrStProzessData^.rCentringOffsetSlowToFastZSpeed:=STRING_TO_REAL(sValue); iCountParameter:=iCountParameter + 1;
		ELSIF sVariableName = 'icentringselectprocess' THEN ptrStProzessData^.iCentringSelectProcess:=STRING_TO_INT(sValue); iCountParameter:=iCountParameter + 1;
		ELSIF sVariableName = 'xpositionendprocinconoff' THEN ptrStProzessData^.xPositionEndProcIncOnOff:=STRING_TO_BOOL(sValue); iCountParameter:=iCountParameter + 1;
		ELSIF sVariableName = 'rpositionendprocmaxinc' THEN ptrStProzessData^.rPositionEndProcMaxInc:=STRING_TO_REAL(sValue); iCountParameter:=iCountParameter + 1;
		ELSIF sVariableName = 'rpositionendproinc' THEN ptrStProzessData^.rPositionEndProInc:=STRING_TO_REAL(sValue); iCountParameter:=iCountParameter + 1;
		ELSIF sVariableName = 'routfeedstrokeaxisspeedslow' THEN ptrStProzessData^.rOutfeedStrokeAxisSpeedSlow:=STRING_TO_REAL(sValue); iCountParameter:=iCountParameter + 1;
		ELSIF sVariableName = 'rz1axisposswitchfastvel' THEN ptrStProzessData^.rZ1AxisPosSwitchFastVel:=STRING_TO_REAL(sValue); iCountParameter:=iCountParameter + 1;
		ELSIF sVariableName = 'rz1axisoffsetstartrecordtorque' THEN ptrStProzessData^.rZ1AxisOffsetStartRecordTorque:=STRING_TO_REAL(sValue); iCountParameter:=iCountParameter + 1;
		ELSIF sVariableName = 'xcentringendprocinconoff' THEN ptrStProzessData^.xCentringEndProcIncOnOff:=STRING_TO_BOOL(sValue); iCountParameter:=iCountParameter + 1;
		ELSIF sVariableName = 'rcentringendproinc' THEN ptrStProzessData^.rCentringEndProInc:=STRING_TO_REAL(sValue); iCountParameter:=iCountParameter + 1;
		ELSIF sVariableName = 'rworkingspindlespeedminmax' THEN ptrStProzessData^.rWorkingSpindleSpeedMinMax:=STRING_TO_REAL(sValue); iCountParameter:=iCountParameter + 1;
		ELSIF sVariableName = 'ro_ctrl_torquepercent_off' THEN ptrStProzessData^.rO_Ctrl_TorquePercent_OFF:=STRING_TO_REAL(sValue); iCountParameter:=iCountParameter + 1;
		ELSIF sVariableName = 'ro_ctrl_hystereseoffset' THEN ptrStProzessData^.rO_Ctrl_HystereseOffset:=STRING_TO_REAL(sValue); iCountParameter:=iCountParameter + 1;
		ELSIF sVariableName = 'rzpositioncylindricalarea' THEN ptrStProzessData^.rZPositionCylindricalArea:=STRING_TO_REAL(sValue); iCountParameter:=iCountParameter + 1;
		ELSIF sVariableName = 'rzminthresholdtroqueendprocess' THEN ptrStProzessData^.rZMinThresholdTroqueEndProcess:=STRING_TO_REAL(sValue); iCountParameter:=iCountParameter + 1;

		ELSIF sVariableName = 'iworkcontroltype' THEN ptrStProzessData^.iWorkControlType:=STRING_TO_INT(sValue); iCountParameter:=iCountParameter + 1;
		ELSIF sVariableName = 'rz_pid_torque' THEN ptrStProzessData^.rZ_PID_Torque:=STRING_TO_REAL(sValue); iCountParameter:=iCountParameter + 1;
		ELSIF sVariableName = 'rz_pid_minspeed' THEN ptrStProzessData^.rZ_PID_MinSpeed:=STRING_TO_REAL(sValue); iCountParameter:=iCountParameter + 1;
		ELSIF sVariableName = 'rz_pid_maxspeed' THEN ptrStProzessData^.rZ_PID_MaxSpeed:=STRING_TO_REAL(sValue); iCountParameter:=iCountParameter + 1;
		ELSIF sVariableName = 'rz_pid_kp' THEN ptrStProzessData^.rZ_PID_Kp:=STRING_TO_REAL(sValue); iCountParameter:=iCountParameter + 1;
		ELSIF sVariableName = 'rz_pid_ki' THEN ptrStProzessData^.rZ_PID_Ki:=STRING_TO_REAL(sValue); iCountParameter:=iCountParameter + 1;
		ELSIF sVariableName = 'rz_pid_kd' THEN ptrStProzessData^.rZ_PID_Kd:=STRING_TO_REAL(sValue); iCountParameter:=iCountParameter + 1;
		ELSIF sVariableName = 'iz_pid_filterm' THEN ptrStProzessData^.iZ_PID_FilterM:=STRING_TO_INT(sValue); iCountParameter:=iCountParameter + 1;
		ELSIF sVariableName = 'rz_d_kd' THEN ptrStProzessData^.rZ_D_Kd:=STRING_TO_REAL(sValue); iCountParameter:=iCountParameter + 1;
		ELSIF sVariableName = 'iz_d_filterm' THEN ptrStProzessData^.iZ_D_FilterM:=STRING_TO_INT(sValue); iCountParameter:=iCountParameter + 1;

		ELSIF sVariableName = 'rsuspensionbubblerspeed' THEN ptrStProzessData^.rSuspensionBubblerSpeed:=STRING_TO_REAL(sValue); iCountParameter:=iCountParameter + 1;
		ELSIF sVariableName = 'rsuspensionfeederspeed' THEN ptrStProzessData^.rSuspensionFeederSpeed:=STRING_TO_REAL(sValue); iCountParameter:=iCountParameter + 1;

		ELSIF sVariableName = 'rdistprogressstroke' THEN ptrStProzessData^.rDistProgressStroke:=STRING_TO_REAL(sValue); iCountParameter:=iCountParameter + 1;
		ELSIF sVariableName = 'iprogressstrokestarttorque' THEN ptrStProzessData^.iProgressStrokeStartTorque:=STRING_TO_INT(sValue); iCountParameter:=iCountParameter + 1;
		ELSIF sVariableName = 'rprogressstrokestopoffset' THEN ptrStProzessData^.rProgressStrokeStopOffset:=STRING_TO_REAL(sValue); iCountParameter:=iCountParameter + 1;
		ELSIF sVariableName = 'icleannozzlemode' THEN ptrStProzessData^.iCleanNozzleMode:=STRING_TO_INT(sValue); iCountParameter:=iCountParameter + 1;
		ELSIF sVariableName = 'ioutfeedstrokecontroller' THEN ptrStProzessData^.iOutfeedStrokeController:=STRING_TO_INT(sValue); iCountParameter:=iCountParameter + 1;
		ELSIF sVariableName = 'isparkoutcontroller' THEN ptrStProzessData^.iSparkOutController:=STRING_TO_INT(sValue); iCountParameter:=iCountParameter + 1;

		END_IF;
	END_IF;
END_IF;
END_ACTION

